KUKA KRL program: EPS_2_25694_LG03A_A_20260223033041.src

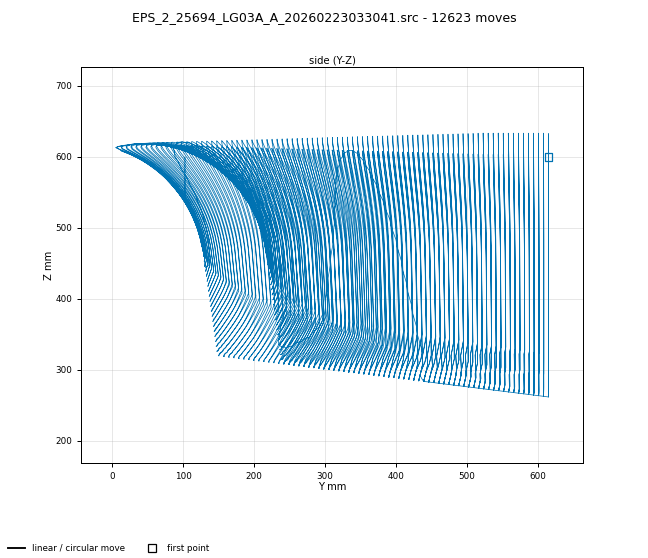
[picture p0: tool path of EPS_2_25694_LG03A_A_20260223033041.src, 12623 of 12625 moves have a stored position in this frame; points joined in program order, loops and branches not executed]
&ACCESS RVP
&REL 4
&COMMENT QRS 19112012
&PARAM EDITMASK = *
DEF PART()
EXT BAS (BAS_COMMAND :IN,REAL :IN )
INT I
BAS (#INITMOV,0 )

;KUKA QRS Post kuka4.cps  Date:22-06-2017 !

File_ID=3042

QRS_PRE_INIT()

;Init var - Until changes are made in qrs_pre_init
Outlet_Square_prg=0
Inlet_1_Square_prg=0
Inlet_2_Square_prg=0
Inlet_3_Square_prg=0
Inlet_4_Square_prg=0
Inlet_5_Square_prg=0

Outlet_1={X 0.000, Y 523.550, Z 484.000, B 0.000, E1 0.000 }
Inlet_1={X 0.000, Y 525.740, Z 454.000, B 0.000, E1 210.000 }
Outlet_1_type=299
Inlet_1_type=299
;QRS#1=Sidecore dimensions
;QRS#2=300-12" PVC SDR 35
;QRS#3=300-12" PVC SDR 35
;QRS#4=
;QRS#5=
;QRS#6=
;QRS#7=
;QRS#8=
;QRS#9=16M PSX
;QRS#10=16M PSX
;QRS#11=
;QRS#12=
;QRS#13=
;QRS#14=
;QRS#15=
;QRS#16=1220x127x914 3'
;QRS#17=EPS Height
;QRS#18=633,5
;QRS#19=*
;QRS#20= UPDATED VERSION 22-06-2017
;QRS#21=*
Outlet_Square=0150
Inlet_1_Square=0150
Inlet_2_Square=0
Inlet_3_Square=0
Inlet_4_Square=0
Inlet_5_Square=0
Mill_Square=1
Outlet_Square_Prg=206
Inlet_1_Square_prg=206

QRS_INIT()

$ADVANCE=5

; T1
PTP {E1 173.663,E2 173.663}
PTP {X 0,Y 615.411,A -85,B 0,C 180,E1 173.663,E2 173.663,E3 0,E4 0,E5 0,E6 0}
QRS_SPEED_INIT()
LIN {X 0,Y 615.411,Z 600,A -85,B 0,C 180,E1 173.663,E2 173.663,E3 0,E4 0,E5 0,E6 0} C_VEL
LIN {X 0,Y 615.411,Z 271.503,A -85,B 0,C 180,E1 173.663,E2 173.663} C_VEL
LIN {X 0,Y 615.411,Z 263.325,A -85,B 0,C 180,E1 173.663,E2 173.663} C_VEL
LIN {X 0,Y 615.409,Z 261.325,A -85,B 0,C 180,E1 173.477,E2 173.477} C_VEL
LIN {X 0,Y 615.462,Z 261.325,A -85,B 0,C 180,E1 170.802,E2 170.802} C_VEL
LIN {X 0,Y 615.44,Z 261.324,A -85,B 0,C 180,E1 168.14,E2 168.14} C_VEL
LIN {X 0,Y 615.434,Z 261.324,A -85,B 0,C 180,E1 166.084,E2 166.084} C_VEL
LIN {X 0,Y 615.412,Z 261.324,A -85,B 0,C 180,E1 163.59,E2 163.59} C_VEL
LIN {X 0,Y 615.421,Z 261.324,A -85,B 0,C 180,E1 161.353,E2 161.353} C_VEL
LIN {X 0,Y 615.489,Z 261.323,A -85,B 0,C 180,E1 158.57,E2 158.57} C_VEL
LIN {X 0,Y 615.417,Z 261.323,A -85,B 0,C 180,E1 155.727,E2 155.727} C_VEL
LIN {X 0,Y 615.419,Z 261.323,A -85,B 0,C 180,E1 153.554,E2 153.554} C_VEL
LIN {X 0,Y 615.479,Z 261.323,A -85,B 0,C 180,E1 150.595,E2 150.595} C_VEL
LIN {X 0,Y 615.45,Z 261.321,A -85,B 0,C 180,E1 148.314,E2 148.314} C_VEL
LIN {X 0,Y 615.424,Z 261.322,A -85,B 0,C 180,E1 145.976,E2 145.976} C_VEL
LIN {X 0,Y 615.426,Z 261.323,A -85,B 0,C 180,E1 143.573,E2 143.573} C_VEL
LIN {X 0,Y 615.491,Z 261.325,A -85,B 0,C 180,E1 140.936,E2 140.936} C_VEL
LIN {X 0,Y 615.47,Z 261.319,A -85,B 0,C 180,E1 138.527,E2 138.527} C_VEL
LIN {X 0,Y 615.425,Z 261.321,A -85,B 0,C 180,E1 136.008,E2 136.008} C_VEL
LIN {X 0,Y 615.428,Z 261.321,A -85,B 0,C 180,E1 133.994,E2 133.994} C_VEL
LIN {X 0,Y 615.442,Z 261.323,A -85,B 0,C 180,E1 131.477,E2 131.477} C_VEL
LIN {X 0,Y 615.495,Z 261.322,A -85,B 0,C 180,E1 128.903,E2 128.903} C_VEL
LIN {X 0,Y 615.453,Z 261.318,A -85,B 0,C 180,E1 126.426,E2 126.426} C_VEL
LIN {X 0,Y 615.431,Z 261.32,A -85,B 0,C 180,E1 124.025,E2 124.025} C_VEL
LIN {X 0,Y 615.487,Z 261.328,A -85,B 0,C 180,E1 121.09,E2 121.09} C_VEL
LIN {X 0,Y 615.45,Z 261.318,A -85,B 0,C 180,E1 118.448,E2 118.448} C_VEL
LIN {X 0,Y 615.452,Z 261.317,A -85,B 0,C 180,E1 116.445,E2 116.445} C_VEL
LIN {X 0,Y 615.435,Z 261.32,A -85,B 0,C 180,E1 114.002,E2 114.002} C_VEL
LIN {X 0,Y 615.47,Z 261.324,A -85,B 0,C 180,E1 111.432,E2 111.432} C_VEL
LIN {X 0,Y 615.464,Z 261.315,A -85,B 0,C 180,E1 108.605,E2 108.605} C_VEL
LIN {X 0,Y 615.449,Z 261.317,A -85,B 0,C 180,E1 106.426,E2 106.426} C_VEL
LIN {X 0,Y 615.444,Z 261.321,A -85,B 0,C 180,E1 103.875,E2 103.875} C_VEL
LIN {X 0,Y 615.484,Z 261.315,A -85,B 0,C 180,E1 100.898,E2 100.898} C_VEL
LIN {X 0,Y 615.455,Z 261.315,A -85,B 0,C 180,E1 98.537,E2 98.537} C_VEL
LIN {X 0,Y 615.456,Z 261.315,A -85,B 0,C 180,E1 96.557,E2 96.557} C_VEL
LIN {X 0,Y 615.456,Z 261.315,A -85,B 0,C 180,E1 94.585,E2 94.585} C_VEL
LIN {X 0,Y 615.46,Z 261.314,A -85,B 0,C 180,E1 92.618,E2 92.618} C_VEL
LIN {X 0,Y 615.462,Z 261.314,A -85,B 0,C 180,E1 90.655,E2 90.655} C_VEL
LIN {X 0,Y 615.447,Z 261.32,A -85,B 0,C 180,E1 88.037,E2 88.037} C_VEL
LIN {X 0,Y 615.497,Z 261.323,A -85,B 0,C 180,E1 85.416,E2 85.416} C_VEL
LIN {X 0,Y 615.471,Z 261.312,A -85,B 0,C 180,E1 82.785,E2 82.785} C_VEL
LIN {X 0,Y 615.448,Z 261.483,A -85,B 0,C 180,E1 82.248,E2 82.248} C_VEL
LIN {X 0,Y 615.472,Z 281.565,A -85,B 0,C 180,E1 79.64,E2 79.64} C_VEL
LIN {X 0,Y 615.452,Z 293.149,A -85,B 0,C 180,E1 78.181,E2 78.181} C_VEL
LIN {X 0,Y 615.487,Z 458.004,A -85,B 0,C 180,E1 76.19,E2 76.19} C_VEL
LIN {X 0,Y 615.486,Z 473.487,A -85,B 0,C 180,E1 75.866,E2 75.866} C_VEL
LIN {X 0,Y 615.481,Z 488.594,A -85,B 0,C 180,E1 75.409,E2 75.409} C_VEL
LIN {X 0,Y 615.487,Z 502.357,A -85,B 0,C 180,E1 74.859,E2 74.859} C_VEL
LIN {X 0,Y 615.489,Z 515.954,A -85,B 0,C 180,E1 74.181,E2 74.181} C_VEL
LIN {X 0,Y 615.497,Z 528.53,A -85,B 0,C 180,E1 73.414,E2 73.414} C_VEL
LIN {X 0,Y 615.496,Z 540.263,A -85,B 0,C 180,E1 72.559,E2 72.559} C_VEL
LIN {X 0,Y 615.497,Z 551.874,A -85,B 0,C 180,E1 71.551,E2 71.551} C_VEL
LIN {X 0,Y 615.496,Z 562.114,A -85,B 0,C 180,E1 70.49,E2 70.49} C_VEL
LIN {X 0,Y 615.493,Z 570.715,A -85,B 0,C 180,E1 69.436,E2 69.436} C_VEL
LIN {X 0,Y 615.498,Z 579.036,A -85,B 0,C 180,E1 68.217,E2 68.217} C_VEL
LIN {X 0,Y 615.494,Z 585.106,A -85,B 0,C 180,E1 67.157,E2 67.157} C_VEL
LIN {X 0,Y 615.492,Z 590.575,A -85,B 0,C 180,E1 65.986,E2 65.986} C_VEL
LIN {X 0,Y 615.498,Z 594.352,A -85,B 0,C 180,E1 65.01,E2 65.01} C_VEL
LIN {X 0,Y 615.49,Z 598.605,A -85,B 0,C 180,E1 63.557,E2 63.557} C_VEL
LIN {X 0,Y 615.493,Z 601.396,A -85,B 0,C 180,E1 62.086,E2 62.086} C_VEL
LIN {X 0,Y 615.496,Z 602.743,A -85,B 0,C 180,E1 60.595,E2 60.595} C_VEL
LIN {X 0,Y 615.496,Z 602.613,A -85,B 0,C 180,E1 59.082,E2 59.082} C_VEL
LIN {X 0,Y 615.49,Z 601.149,A -85,B 0,C 180,E1 57.665,E2 57.665} C_VEL
LIN {X 0,Y 615.491,Z 598.842,A -85,B 0,C 180,E1 56.462,E2 56.462} C_VEL
LIN {X 0,Y 615.499,Z 595.27,A -85,B 0,C 180,E1 55.187,E2 55.187} C_VEL
LIN {X 0,Y 615.497,Z 590.342,A -85,B 0,C 180,E1 53.87,E2 53.87} C_VEL
LIN {X 0,Y 615.497,Z 584.083,A -85,B 0,C 180,E1 52.567,E2 52.567} C_VEL
LIN {X 0,Y 615.493,Z 576.583,A -85,B 0,C 180,E1 51.307,E2 51.307} C_VEL
LIN {X 0,Y 615.494,Z 567.668,A -85,B 0,C 180,E1 50.08,E2 50.08} C_VEL
LIN {X 0,Y 615.494,Z 558.54,A -85,B 0,C 180,E1 49.026,E2 49.026} C_VEL
LIN {X 0,Y 615.494,Z 548.798,A -85,B 0,C 180,E1 48.07,E2 48.07} C_VEL
LIN {X 0,Y 615.496,Z 537.414,A -85,B 0,C 180,E1 47.125,E2 47.125} C_VEL
LIN {X 0,Y 615.498,Z 525.333,A -85,B 0,C 180,E1 46.285,E2 46.285} C_VEL
LIN {X 0,Y 615.485,Z 512.772,A -85,B 0,C 180,E1 45.558,E2 45.558} C_VEL
LIN {X 0,Y 615.493,Z 499.631,A -85,B 0,C 180,E1 44.934,E2 44.934} C_VEL
LIN {X 0,Y 615.49,Z 485.257,A -85,B 0,C 180,E1 44.392,E2 44.392} C_VEL
LIN {X 0,Y 615.492,Z 469.545,A -85,B 0,C 180,E1 43.952,E2 43.952} C_VEL
LIN {X 0,Y 615.492,Z 454.254,A -85,B 0,C 180,E1 43.667,E2 43.667} C_VEL
LIN {X 0,Y 615.466,Z 292.857,A -85,B 0,C 180,E1 41.719,E2 41.719} C_VEL
LIN {X 0,Y 615.478,Z 270.989,A -85,B 0,C 180,E1 38.903,E2 38.903} C_VEL
LIN {X 0,Y 615.477,Z 261.311,A -85,B 0,C 180,E1 37.626,E2 37.626} C_VEL
LIN {X 0,Y 615.484,Z 261.319,A -85,B 0,C 180,E1 34.702,E2 34.702} C_VEL
LIN {X 0,Y 615.486,Z 261.323,A -85,B 0,C 180,E1 32.333,E2 32.333} C_VEL
LIN {X 0,Y 615.485,Z 261.308,A -85,B 0,C 180,E1 29.405,E2 29.405} C_VEL
LIN {X 0,Y 615.482,Z 261.324,A -85,B 0,C 180,E1 26.443,E2 26.443} C_VEL
LIN {X 0,Y 615.482,Z 261.309,A -85,B 0,C 180,E1 23.555,E2 23.555} C_VEL
LIN {X 0,Y 615.481,Z 261.324,A -85,B 0,C 180,E1 20.559,E2 20.559} C_VEL
LIN {X 0,Y 615.46,Z 261.315,A -85,B 0,C 180,E1 17.956,E2 17.956} C_VEL
LIN {X 0,Y 615.492,Z 261.313,A -85,B 0,C 180,E1 15.225,E2 15.225} C_VEL
LIN {X 0,Y 615.469,Z 261.321,A -85,B 0,C 180,E1 12.529,E2 12.529} C_VEL
LIN {X 0,Y 615.461,Z 261.314,A -85,B 0,C 180,E1 9.861,E2 9.861} C_VEL
LIN {X 0,Y 615.494,Z 261.317,A -85,B 0,C 180,E1 7.214,E2 7.214} C_VEL
LIN {X 0,Y 615.459,Z 261.321,A -85,B 0,C 180,E1 4.584,E2 4.584} C_VEL
LIN {X 0,Y 615.454,Z 261.315,A -85,B 0,C 180,E1 1.962,E2 1.962} C_VEL
LIN {X 0,Y 615.494,Z 261.317,A -85,B 0,C 180,E1 -0.655,E2 -0.655} C_VEL
LIN {X 0,Y 615.454,Z 261.322,A -85,B 0,C 180,E1 -3.274,E2 -3.274} C_VEL
LIN {X 0,Y 615.454,Z 261.322,A -85,B 0,C 180,E1 -5.242,E2 -5.242} C_VEL
LIN {X 0,Y 615.452,Z 261.323,A -85,B 0,C 180,E1 -7.217,E2 -7.217} C_VEL
LIN {X 0,Y 615.45,Z 261.323,A -85,B 0,C 180,E1 -9.2,E2 -9.2} C_VEL
LIN {X 0,Y 615.447,Z 261.322,A -85,B 0,C 180,E1 -11.195,E2 -11.195} C_VEL
LIN {X 0,Y 615.443,Z 261.322,A -85,B 0,C 180,E1 -13.203,E2 -13.203} C_VEL
LIN {X 0,Y 615.438,Z 261.322,A -85,B 0,C 180,E1 -15.228,E2 -15.228} C_VEL
LIN {X 0,Y 615.433,Z 261.322,A -85,B 0,C 180,E1 -17.273,E2 -17.273} C_VEL
LIN {X 0,Y 615.427,Z 261.322,A -85,B 0,C 180,E1 -19.341,E2 -19.341} C_VEL
LIN {X 0,Y 615.423,Z 261.322,A -85,B 0,C 180,E1 -21.435,E2 -21.435} C_VEL
LIN {X 0,Y 615.446,Z 261.322,A -85,B 0,C 180,E1 -24.003,E2 -24.003} C_VEL
LIN {X 0,Y 615.492,Z 261.327,A -85,B 0,C 180,E1 -26.445,E2 -26.445} C_VEL
LIN {X 0,Y 615.462,Z 261.325,A -85,B 0,C 180,E1 -28.66,E2 -28.66} C_VEL
LIN {X 0,Y 615.419,Z 261.325,A -85,B 0,C 180,E1 -31.078,E2 -31.078} C_VEL
LIN {X 0,Y 615.411,Z 261.325,A -85,B 0,C 180,E1 -33.241,E2 -33.241} C_VEL
LIN {X 0,Y 615.435,Z 261.326,A -85,B 0,C 180,E1 -35.829,E2 -35.829} C_VEL
LIN {X 0,Y 615.473,Z 261.325,A -85,B 0,C 180,E1 -38.07,E2 -38.07} C_VEL
LIN {X 0,Y 615.452,Z 261.323,A -85,B 0,C 180,E1 -40.61,E2 -40.61} C_VEL
LIN {X 0,Y 615.422,Z 261.323,A -85,B 0,C 180,E1 -43.043,E2 -43.043} C_VEL
LIN {X 0,Y 615.422,Z 261.322,A -85,B 0,C 180,E1 -45.075,E2 -45.075} C_VEL
LIN {X 0,Y 615.446,Z 261.324,A -85,B 0,C 180,E1 -47.645,E2 -47.645} C_VEL
LIN {X 0,Y 615.491,Z 261.319,A -85,B 0,C 180,E1 -50.252,E2 -50.252} C_VEL
LIN {X 0,Y 615.439,Z 261.32,A -85,B 0,C 180,E1 -52.756,E2 -52.756} C_VEL
LIN {X 0,Y 615.431,Z 261.322,A -85,B 0,C 180,E1 -55.183,E2 -55.183} C_VEL
LIN {X 0,Y 615.472,Z 261.324,A -85,B 0,C 180,E1 -57.672,E2 -57.672} C_VEL
LIN {X 0,Y 615.452,Z 261.317,A -85,B 0,C 180,E1 -60.593,E2 -60.593} C_VEL
LIN {X 0,Y 615.439,Z 261.319,A -85,B 0,C 180,E1 -62.964,E2 -62.964} C_VEL
LIN {X 0,Y 615.441,Z 261.447,A -85,B 0,C 180,E1 -64.936,E2 -64.936} C_VEL
LIN {X 0,Y 615.482,Z 284.085,A -85,B 0,C 180,E1 -67.53,E2 -67.53} C_VEL
LIN {X 0,Y 615.49,Z 308.883,A -85,B 0,C 180,E1 -70.316,E2 -70.316} C_VEL
LIN {X 0,Y 615.488,Z 322.077,A -85,B 0,C 180,E1 -71.762,E2 -71.762} C_VEL
LIN {X 0,Y 615.487,Z 488.142,A -85,B 0,C 180,E1 -73.768,E2 -73.768} C_VEL
LIN {X 0,Y 615.49,Z 503.738,A -85,B 0,C 180,E1 -74.096,E2 -74.096} C_VEL
LIN {X 0,Y 615.48,Z 519.068,A -85,B 0,C 180,E1 -74.562,E2 -74.562} C_VEL
LIN {X 0,Y 615.492,Z 532.768,A -85,B 0,C 180,E1 -75.113,E2 -75.113} C_VEL
LIN {X 0,Y 615.494,Z 547.053,A -85,B 0,C 180,E1 -75.834,E2 -75.834} C_VEL
LIN {X 0,Y 615.497,Z 559.907,A -85,B 0,C 180,E1 -76.632,E2 -76.632} C_VEL
LIN {X 0,Y 615.495,Z 572.262,A -85,B 0,C 180,E1 -77.554,E2 -77.554} C_VEL
LIN {X 0,Y 615.495,Z 582.612,A -85,B 0,C 180,E1 -78.474,E2 -78.474} C_VEL
LIN {X 0,Y 615.495,Z 592.189,A -85,B 0,C 180,E1 -79.474,E2 -79.474} C_VEL
LIN {X 0,Y 615.494,Z 601.581,A -85,B 0,C 180,E1 -80.636,E2 -80.636} C_VEL
LIN {X 0,Y 615.495,Z 609.384,A -85,B 0,C 180,E1 -81.795,E2 -81.795} C_VEL
LIN {X 0,Y 615.496,Z 616.608,A -85,B 0,C 180,E1 -83.102,E2 -83.102} C_VEL
LIN {X 0,Y 615.499,Z 622.438,A -85,B 0,C 180,E1 -84.431,E2 -84.431} C_VEL
LIN {X 0,Y 615.491,Z 625.861,A -85,B 0,C 180,E1 -85.416,E2 -85.416} C_VEL
LIN {X 0,Y 615.492,Z 629.319,A -85,B 0,C 180,E1 -86.727,E2 -86.727} C_VEL
LIN {X 0,Y 615.497,Z 631.594,A -85,B 0,C 180,E1 -88.037,E2 -88.037} C_VEL
LIN {X 0,Y 615.493,Z 632.741,A -85,B 0,C 180,E1 -89.346,E2 -89.346} C_VEL
LIN {X 0,Y 615.493,Z 632.74,A -85,B 0,C 180,E1 -90.654,E2 -90.654} C_VEL
LIN {X 0,Y 615.497,Z 631.593,A -85,B 0,C 180,E1 -91.963,E2 -91.963} C_VEL
LIN {X 0,Y 615.492,Z 629.318,A -85,B 0,C 180,E1 -93.273,E2 -93.273} C_VEL
LIN {X 0,Y 615.491,Z 625.86,A -85,B 0,C 180,E1 -94.585,E2 -94.585} C_VEL
LIN {X 0,Y 615.49,Z 621.143,A -85,B 0,C 180,E1 -95.899,E2 -95.899} C_VEL
LIN {X 0,Y 615.495,Z 615.029,A -85,B 0,C 180,E1 -97.216,E2 -97.216} C_VEL
LIN {X 0,Y 615.49,Z 607.332,A -85,B 0,C 180,E1 -98.537,E2 -98.537} C_VEL
LIN {X 0,Y 615.495,Z 599.113,A -85,B 0,C 180,E1 -99.696,E2 -99.696} C_VEL
LIN {X 0,Y 615.497,Z 588.897,A -85,B 0,C 180,E1 -100.892,E2 -100.892} C_VEL
LIN {X 0,Y 615.495,Z 579.067,A -85,B 0,C 180,E1 -101.861,E2 -101.861} C_VEL
LIN {X 0,Y 615.498,Z 566.947,A -85,B 0,C 180,E1 -102.865,E2 -102.865} C_VEL
LIN {X 0,Y 615.498,Z 554.798,A -85,B 0,C 180,E1 -103.705,E2 -103.705} C_VEL
LIN {X 0,Y 615.484,Z 541.38,A -85,B 0,C 180,E1 -104.472,E2 -104.472} C_VEL
LIN {X 0,Y 615.495,Z 526.849,A -85,B 0,C 180,E1 -105.141,E2 -105.141} C_VEL
LIN {X 0,Y 615.484,Z 512.618,A -85,B 0,C 180,E1 -105.65,E2 -105.65} C_VEL
LIN {X 0,Y 615.499,Z 498.131,A -85,B 0,C 180,E1 -106.036,E2 -106.036} C_VEL
LIN {X 0,Y 615.487,Z 483.544,A -85,B 0,C 180,E1 -106.298,E2 -106.298} C_VEL
LIN {X 0,Y 615.489,Z 321.745,A -85,B 0,C 180,E1 -108.258,E2 -108.258} C_VEL
LIN {X 0,Y 615.49,Z 296.393,A -85,B 0,C 180,E1 -111.081,E2 -111.081} C_VEL
LIN {X 0,Y 615.495,Z 270.582,A -85,B 0,C 180,E1 -114.01,E2 -114.01} C_VEL
LIN {X 0,Y 615.441,Z 261.318,A -85,B 0,C 180,E1 -115.1,E2 -115.1} C_VEL
LIN {X 0,Y 615.489,Z 261.317,A -85,B 0,C 180,E1 -117.915,E2 -117.915} C_VEL
LIN {X 0,Y 615.498,Z 261.324,A -85,B 0,C 180,E1 -120.159,E2 -120.159} C_VEL
LIN {X 0,Y 615.465,Z 261.323,A -85,B 0,C 180,E1 -122.458,E2 -122.458} C_VEL
LIN {X 0,Y 615.439,Z 261.32,A -85,B 0,C 180,E1 -124.818,E2 -124.818} C_VEL
LIN {X 0,Y 615.443,Z 261.318,A -85,B 0,C 180,E1 -127.245,E2 -127.245} C_VEL
LIN {X 0,Y 615.498,Z 261.326,A -85,B 0,C 180,E1 -130.09,E2 -130.09} C_VEL
LIN {X 0,Y 615.463,Z 261.323,A -85,B 0,C 180,E1 -132.354,E2 -132.354} C_VEL
LIN {X 0,Y 615.433,Z 261.32,A -85,B 0,C 180,E1 -134.926,E2 -134.926} C_VEL
LIN {X 0,Y 615.433,Z 261.32,A -85,B 0,C 180,E1 -136.957,E2 -136.957} C_VEL
LIN {X 0,Y 615.457,Z 261.317,A -85,B 0,C 180,E1 -139.391,E2 -139.391} C_VEL
LIN {X 0,Y 615.481,Z 261.328,A -85,B 0,C 180,E1 -141.988,E2 -141.988} C_VEL
LIN {X 0,Y 615.446,Z 261.323,A -85,B 0,C 180,E1 -144.381,E2 -144.381} C_VEL
LIN {X 0,Y 615.428,Z 261.321,A -85,B 0,C 180,E1 -146.76,E2 -146.76} C_VEL
LIN {X 0,Y 615.435,Z 261.32,A -85,B 0,C 180,E1 -149.077,E2 -149.077} C_VEL
LIN {X 0,Y 615.484,Z 261.318,A -85,B 0,C 180,E1 -151.549,E2 -151.549} C_VEL
LIN {X 0,Y 615.443,Z 261.323,A -85,B 0,C 180,E1 -154.282,E2 -154.282} C_VEL
LIN {X 0,Y 615.43,Z 261.323,A -85,B 0,C 180,E1 -156.441,E2 -156.441} C_VEL
LIN {X 0,Y 615.424,Z 261.323,A -85,B 0,C 180,E1 -158.565,E2 -158.565} C_VEL
LIN {X 0,Y 615.422,Z 261.322,A -85,B 0,C 180,E1 -160.659,E2 -160.659} C_VEL
LIN {X 0,Y 615.47,Z 261.321,A -85,B 0,C 180,E1 -163.412,E2 -163.412} C_VEL
LIN {X 0,Y 615.443,Z 261.324,A -85,B 0,C 180,E1 -166.124,E2 -166.124} C_VEL
LIN {X 0,Y 615.44,Z 261.324,A -85,B 0,C 180,E1 -168.137,E2 -168.137} C_VEL
LIN {X 0,Y 615.437,Z 261.324,A -85,B 0,C 180,E1 -170.136,E2 -170.136} C_VEL
LIN {X 0,Y 615.436,Z 261.324,A -85,B 0,C 180,E1 -172.123,E2 -172.123} C_VEL
LIN {X 0,Y 615.436,Z 261.324,A -85,B 0,C 180,E1 -174.1,E2 -174.1} C_VEL
LIN {X 0,Y 615.436,Z 261.324,A -85,B 0,C 180,E1 -176.07,E2 -176.07} C_VEL
LIN {X 0,Y 615.437,Z 261.325,A -85,B 0,C 180,E1 -178.036,E2 -178.036} C_VEL
LIN {X 0,Y 615.437,Z 261.325,A -85,B 0,C 180,E1 -179.999,E2 -179.999} C_VEL
LIN {X 0,Y 615.439,Z 261.325,A -85,B 0,C 180,E1 -181.962,E2 -181.962} C_VEL
LIN {X 0,Y 615.44,Z 261.325,A -85,B 0,C 180,E1 -183.928,E2 -183.928} C_VEL
LIN {X 0,Y 615.409,Z 261.325,A -85,B 0,C 180,E1 -186.523,E2 -186.523} C_VEL
LIN {X 0,Y 614.767,Z 261.474,A -85,B 0,C 180,E1 -187.069,E2 -187.069} C_VEL
LIN {X 0,Y 611.966,Z 261.877,A -85,B 0,C 180,E1 -187.955,E2 -187.955} C_VEL
LIN {X 0,Y 609.577,Z 262.192,A -85,B 0,C 180,E1 -188.668,E2 -188.668} C_VEL
LIN {X 0,Y 608.529,Z 262.313,A -85,B 0,C 180,E1 -189.218,E2 -189.218} C_VEL
LIN {X 0,Y 608.433,Z 262.321,A -85,B 0,C 180,E1 -189.404,E2 -189.404} C_VEL
LIN {X 0,Y 608.414,Z 262.319,A -85,B 0,C 180,E1 -191.999,E2 -191.999} C_VEL
LIN {X 0,Y 608.405,Z 262.319,A -85,B 0,C 180,E1 -194.038,E2 -194.038} C_VEL
LIN {X 0,Y 608.384,Z 262.32,A -85,B 0,C 180,E1 -196.506,E2 -196.506} C_VEL
LIN {X 0,Y 608.423,Z 262.319,A -85,B 0,C 180,E1 -198.869,E2 -198.869} C_VEL
LIN {X 0,Y 608.445,Z 262.317,A -85,B 0,C 180,E1 -201.691,E2 -201.691} C_VEL
LIN {X 0,Y 608.408,Z 262.319,A -85,B 0,C 180,E1 -204.571,E2 -204.571} C_VEL
LIN {X 0,Y 608.467,Z 262.32,A -85,B 0,C 180,E1 -207.207,E2 -207.207} C_VEL
LIN {X 0,Y 608.402,Z 262.319,A -85,B 0,C 180,E1 -209.962,E2 -209.962} C_VEL
LIN {X 0,Y 608.415,Z 262.317,A -85,B 0,C 180,E1 -212.095,E2 -212.095} C_VEL
LIN {X 0,Y 608.417,Z 262.323,A -85,B 0,C 180,E1 -214.902,E2 -214.902} C_VEL
LIN {X 0,Y 608.433,Z 262.316,A -85,B 0,C 180,E1 -217.747,E2 -217.747} C_VEL
LIN {X 0,Y 608.414,Z 262.318,A -85,B 0,C 180,E1 -220.326,E2 -220.326} C_VEL
LIN {X 0,Y 608.443,Z 262.322,A -85,B 0,C 180,E1 -222.958,E2 -222.958} C_VEL
LIN {X 0,Y 608.413,Z 262.318,A -85,B 0,C 180,E1 -225.738,E2 -225.738} C_VEL
LIN {X 0,Y 608.413,Z 262.317,A -85,B 0,C 180,E1 -227.935,E2 -227.935} C_VEL
LIN {X 0,Y 608.43,Z 262.321,A -85,B 0,C 180,E1 -230.704,E2 -230.704} C_VEL
LIN {X 0,Y 608.46,Z 262.32,A -85,B 0,C 180,E1 -233.086,E2 -233.086} C_VEL
LIN {X 0,Y 608.452,Z 262.314,A -85,B 0,C 180,E1 -235.53,E2 -235.53} C_VEL
LIN {X 0,Y 608.425,Z 262.316,A -85,B 0,C 180,E1 -237.904,E2 -237.904} C_VEL
LIN {X 0,Y 608.421,Z 262.317,A -85,B 0,C 180,E1 -240.218,E2 -240.218} C_VEL
LIN {X 0,Y 608.477,Z 262.319,A -85,B 0,C 180,E1 -242.789,E2 -242.789} C_VEL
LIN {X 0,Y 608.435,Z 262.314,A -85,B 0,C 180,E1 -245.852,E2 -245.852} C_VEL
LIN {X 0,Y 608.44,Z 262.317,A -85,B 0,C 180,E1 -248.308,E2 -248.308} C_VEL
LIN {X 0,Y 608.451,Z 262.315,A -85,B 0,C 180,E1 -251.283,E2 -251.283} C_VEL
LIN {X 0,Y 608.42,Z 262.316,A -85,B 0,C 180,E1 -253.905,E2 -253.905} C_VEL
LIN {X 0,Y 608.461,Z 262.321,A -85,B 0,C 180,E1 -256.644,E2 -256.644} C_VEL
LIN {X 0,Y 608.443,Z 262.315,A -85,B 0,C 180,E1 -259.35,E2 -259.35} C_VEL
LIN {X 0,Y 608.444,Z 262.315,A -85,B 0,C 180,E1 -262.033,E2 -262.033} C_VEL
LIN {X 0,Y 608.469,Z 262.32,A -85,B 0,C 180,E1 -264.698,E2 -264.698} C_VEL
LIN {X 0,Y 608.453,Z 262.313,A -85,B 0,C 180,E1 -267.352,E2 -267.352} C_VEL
LIN {X 0,Y 608.442,Z 262.316,A -85,B 0,C 180,E1 -270,E2 -270} C_VEL
LIN {X 0,Y 608.484,Z 262.317,A -85,B 0,C 180,E1 -272.648,E2 -272.648} C_VEL
LIN {X 0,Y 608.446,Z 262.314,A -85,B 0,C 180,E1 -275.302,E2 -275.302} C_VEL
LIN {X 0,Y 608.431,Z 262.317,A -85,B 0,C 180,E1 -277.591,E2 -277.591} C_VEL
LIN {X 0,Y 608.559,Z 276.552,A -85,B 0,C 180,E1 -279.472,E2 -279.472} C_VEL
LIN {X 0,Y 608.519,Z 292.986,A -85,B 0,C 180,E1 -281.602,E2 -281.602} C_VEL
LIN {X 0,Y 608.721,Z 316.53,A -85,B 0,C 180,E1 -281.895,E2 -281.895} C_VEL
LIN {X 0,Y 608.666,Z 458.242,A -85,B 0,C 180,E1 -283.628,E2 -283.628} C_VEL
LIN {X 0,Y 608.667,Z 474.141,A -85,B 0,C 180,E1 -283.968,E2 -283.968} C_VEL
LIN {X 0,Y 608.618,Z 489.893,A -85,B 0,C 180,E1 -284.46,E2 -284.46} C_VEL
LIN {X 0,Y 608.596,Z 504.382,A -85,B 0,C 180,E1 -285.059,E2 -285.059} C_VEL
LIN {X 0,Y 608.562,Z 517.647,A -85,B 0,C 180,E1 -285.746,E2 -285.746} C_VEL
LIN {X 0,Y 608.546,Z 530.554,A -85,B 0,C 180,E1 -286.561,E2 -286.561} C_VEL
LIN {X 0,Y 608.508,Z 542.604,A -85,B 0,C 180,E1 -287.474,E2 -287.474} C_VEL
LIN {X 0,Y 608.493,Z 553.997,A -85,B 0,C 180,E1 -288.503,E2 -288.503} C_VEL
LIN {X 0,Y 608.467,Z 563.931,A -85,B 0,C 180,E1 -289.569,E2 -289.569} C_VEL
LIN {X 0,Y 608.46,Z 573.467,A -85,B 0,C 180,E1 -290.79,E2 -290.79} C_VEL
LIN {X 0,Y 608.453,Z 581.573,A -85,B 0,C 180,E1 -292.048,E2 -292.048} C_VEL
LIN {X 0,Y 608.434,Z 587.306,A -85,B 0,C 180,E1 -293.124,E2 -293.124} C_VEL
LIN {X 0,Y 608.427,Z 591.904,A -85,B 0,C 180,E1 -294.147,E2 -294.147} C_VEL
LIN {X 0,Y 608.437,Z 596.043,A -85,B 0,C 180,E1 -295.301,E2 -295.301} C_VEL
LIN {X 0,Y 608.422,Z 599.973,A -85,B 0,C 180,E1 -296.775,E2 -296.775} C_VEL
LIN {X 0,Y 608.434,Z 602.436,A -85,B 0,C 180,E1 -298.267,E2 -298.267} C_VEL
LIN {X 0,Y 608.447,Z 603.444,A -85,B 0,C 180,E1 -299.78,E2 -299.78} C_VEL
LIN {X 0,Y 608.435,Z 602.948,A -85,B 0,C 180,E1 -301.317,E2 -301.317} C_VEL
LIN {X 0,Y 608.416,Z 601.474,A -85,B 0,C 180,E1 -302.519,E2 -302.519} C_VEL
LIN {X 0,Y 608.433,Z 598.145,A -85,B 0,C 180,E1 -304.073,E2 -304.073} C_VEL
LIN {X 0,Y 608.425,Z 594.42,A -85,B 0,C 180,E1 -305.278,E2 -305.278} C_VEL
LIN {X 0,Y 608.449,Z 589.516,A -85,B 0,C 180,E1 -306.501,E2 -306.501} C_VEL
LIN {X 0,Y 608.439,Z 583.238,A -85,B 0,C 180,E1 -307.747,E2 -307.747} C_VEL
LIN {X 0,Y 608.469,Z 575.898,A -85,B 0,C 180,E1 -308.943,E2 -308.943} C_VEL
LIN {X 0,Y 608.468,Z 567.519,A -85,B 0,C 180,E1 -310.084,E2 -310.084} C_VEL
LIN {X 0,Y 608.472,Z 558.024,A -85,B 0,C 180,E1 -311.174,E2 -311.174} C_VEL
LIN {X 0,Y 608.498,Z 547.442,A -85,B 0,C 180,E1 -312.199,E2 -312.199} C_VEL
LIN {X 0,Y 608.545,Z 536.009,A -85,B 0,C 180,E1 -313.133,E2 -313.133} C_VEL
LIN {X 0,Y 608.561,Z 523.952,A -85,B 0,C 180,E1 -313.965,E2 -313.965} C_VEL
LIN {X 0,Y 608.568,Z 511.052,A -85,B 0,C 180,E1 -314.703,E2 -314.703} C_VEL
LIN {X 0,Y 608.63,Z 496.659,A -85,B 0,C 180,E1 -315.369,E2 -315.369} C_VEL
LIN {X 0,Y 608.641,Z 482.482,A -85,B 0,C 180,E1 -315.881,E2 -315.881} C_VEL
LIN {X 0,Y 608.669,Z 467.061,A -85,B 0,C 180,E1 -316.291,E2 -316.291} C_VEL
LIN {X 0,Y 608.695,Z 451.014,A -85,B 0,C 180,E1 -316.567,E2 -316.567} C_VEL
LIN {X 0,Y 608.686,Z 293.883,A -85,B 0,C 180,E1 -318.472,E2 -318.472} C_VEL
LIN {X 0,Y 608.511,Z 292.853,A -85,B 0,C 180,E1 -318.5,E2 -318.5} C_VEL
LIN {X 0,Y 608.574,Z 271.809,A -85,B 0,C 180,E1 -321.24,E2 -321.24} C_VEL
LIN {X 0,Y 608.452,Z 262.314,A -85,B 0,C 180,E1 -322.517,E2 -322.517} C_VEL
LIN {X 0,Y 608.471,Z 262.314,A -85,B 0,C 180,E1 -325.089,E2 -325.089} C_VEL
LIN {X 0,Y 608.462,Z 262.315,A -85,B 0,C 180,E1 -327.907,E2 -327.907} C_VEL
LIN {X 0,Y 608.454,Z 262.313,A -85,B 0,C 180,E1 -330.222,E2 -330.222} C_VEL
LIN {X 0,Y 608.474,Z 262.311,A -85,B 0,C 180,E1 -332.791,E2 -332.791} C_VEL
LIN {X 0,Y 608.443,Z 262.324,A -85,B 0,C 180,E1 -335.43,E2 -335.43} C_VEL
LIN {X 0,Y 608.463,Z 262.311,A -85,B 0,C 180,E1 -338.31,E2 -338.31} C_VEL
LIN {X 0,Y 608.462,Z 262.322,A -85,B 0,C 180,E1 -341.282,E2 -341.282} C_VEL
LIN {X 0,Y 608.438,Z 262.315,A -85,B 0,C 180,E1 -343.907,E2 -343.907} C_VEL
LIN {X 0,Y 608.461,Z 262.314,A -85,B 0,C 180,E1 -346.645,E2 -346.645} C_VEL
LIN {X 0,Y 608.451,Z 262.319,A -85,B 0,C 180,E1 -349.351,E2 -349.351} C_VEL
LIN {X 0,Y 608.452,Z 262.312,A -85,B 0,C 180,E1 -352.034,E2 -352.034} C_VEL
LIN {X 0,Y 608.469,Z 262.315,A -85,B 0,C 180,E1 -354.699,E2 -354.699} C_VEL
LIN {X 0,Y 608.452,Z 262.317,A -85,B 0,C 180,E1 -357.353,E2 -357.353} C_VEL
LIN {X 0,Y 608.444,Z 262.313,A -85,B 0,C 180,E1 -360.001,E2 -360.001} C_VEL
LIN {X 0,Y 608.484,Z 262.315,A -85,B 0,C 180,E1 -362.649,E2 -362.649} C_VEL
LIN {X 0,Y 608.433,Z 262.318,A -85,B 0,C 180,E1 -365.303,E2 -365.303} C_VEL
LIN {X 0,Y 608.419,Z 262.319,A -85,B 0,C 180,E1 -367.301,E2 -367.301} C_VEL
LIN {X 0,Y 608.421,Z 262.317,A -85,B 0,C 180,E1 -369.979,E2 -369.979} C_VEL
LIN {X 0,Y 608.47,Z 262.321,A -85,B 0,C 180,E1 -372.678,E2 -372.678} C_VEL
LIN {X 0,Y 608.427,Z 262.316,A -85,B 0,C 180,E1 -375.408,E2 -375.408} C_VEL
LIN {X 0,Y 608.407,Z 262.318,A -85,B 0,C 180,E1 -377.479,E2 -377.479} C_VEL
LIN {X 0,Y 608.406,Z 262.318,A -85,B 0,C 180,E1 -379.573,E2 -379.573} C_VEL
LIN {X 0,Y 608.423,Z 262.316,A -85,B 0,C 180,E1 -381.694,E2 -381.694} C_VEL
LIN {X 0,Y 608.431,Z 262.324,A -85,B 0,C 180,E1 -384.573,E2 -384.573} C_VEL
LIN {X 0,Y 608.405,Z 262.319,A -85,B 0,C 180,E1 -387.197,E2 -387.197} C_VEL
LIN {X 0,Y 608.397,Z 262.321,A -85,B 0,C 180,E1 -389.024,E2 -389.024} C_VEL
LIN {X 0,Y 608.396,Z 262.319,A -85,B 0,C 180,E1 -391.321,E2 -391.321} C_VEL
LIN {X 0,Y 608.415,Z 262.319,A -85,B 0,C 180,E1 -393.729,E2 -393.729} C_VEL
LIN {X 0,Y 608.429,Z 262.323,A -85,B 0,C 180,E1 -396.094,E2 -396.094} C_VEL
LIN {X 0,Y 608.399,Z 262.323,A -85,B 0,C 180,E1 -398.594,E2 -398.594} C_VEL
LIN {X 0,Y 608.389,Z 262.32,A -85,B 0,C 180,E1 -401.183,E2 -401.183} C_VEL
LIN {X 0,Y 608.416,Z 262.317,A -85,B 0,C 180,E1 -403.305,E2 -403.305} C_VEL
LIN {X 0,Y 608.458,Z 262.322,A -85,B 0,C 180,E1 -406.131,E2 -406.131} C_VEL
LIN {X 0,Y 608.406,Z 262.319,A -85,B 0,C 180,E1 -408.821,E2 -408.821} C_VEL
LIN {X 0,Y 608.454,Z 262.319,A -85,B 0,C 180,E1 -411.762,E2 -411.762} C_VEL
LIN {X 0,Y 608.417,Z 262.317,A -85,B 0,C 180,E1 -414.722,E2 -414.722} C_VEL
LIN {X 0,Y 608.425,Z 262.316,A -85,B 0,C 180,E1 -417.12,E2 -417.12} C_VEL
LIN {X 0,Y 608.476,Z 262.317,A -85,B 0,C 180,E1 -420.027,E2 -420.027} C_VEL
LIN {X 0,Y 608.421,Z 262.317,A -85,B 0,C 180,E1 -422.804,E2 -422.804} C_VEL
LIN {X 0,Y 608.448,Z 262.455,A -85,B 0,C 180,E1 -424.746,E2 -424.746} C_VEL
LIN {X 0,Y 608.665,Z 274.55,A -85,B 0,C 180,E1 -426.164,E2 -426.164} C_VEL
LIN {X 0,Y 608.595,Z 297.959,A -85,B 0,C 180,E1 -428.847,E2 -428.847} C_VEL
LIN {X 0,Y 608.574,Z 322.077,A -85,B 0,C 180,E1 -431.548,E2 -431.548} C_VEL
LIN {X 0,Y 608.727,Z 425.97,A -85,B 0,C 180,E1 -432.814,E2 -432.814} C_VEL
LIN {X 0,Y 608.682,Z 488.142,A -85,B 0,C 180,E1 -433.581,E2 -433.581} C_VEL
LIN {X 0,Y 608.65,Z 503.736,A -85,B 0,C 180,E1 -433.912,E2 -433.912} C_VEL
LIN {X 0,Y 608.618,Z 519.067,A -85,B 0,C 180,E1 -434.384,E2 -434.384} C_VEL
LIN {X 0,Y 608.606,Z 532.771,A -85,B 0,C 180,E1 -434.941,E2 -434.941} C_VEL
LIN {X 0,Y 608.575,Z 546.248,A -85,B 0,C 180,E1 -435.625,E2 -435.625} C_VEL
LIN {X 0,Y 608.554,Z 558.673,A -85,B 0,C 180,E1 -436.391,E2 -436.391} C_VEL
LIN {X 0,Y 608.528,Z 571.29,A -85,B 0,C 180,E1 -437.325,E2 -437.325} C_VEL
LIN {X 0,Y 608.496,Z 582.753,A -85,B 0,C 180,E1 -438.34,E2 -438.34} C_VEL
LIN {X 0,Y 608.476,Z 592.393,A -85,B 0,C 180,E1 -439.351,E2 -439.351} C_VEL
LIN {X 0,Y 608.477,Z 601.857,A -85,B 0,C 180,E1 -440.527,E2 -440.527} C_VEL
LIN {X 0,Y 608.455,Z 609.732,A -85,B 0,C 180,E1 -441.699,E2 -441.699} C_VEL
LIN {X 0,Y 608.441,Z 617.089,A -85,B 0,C 180,E1 -443.034,E2 -443.034} C_VEL
LIN {X 0,Y 608.449,Z 622.925,A -85,B 0,C 180,E1 -444.366,E2 -444.366} C_VEL
LIN {X 0,Y 608.427,Z 626.384,A -85,B 0,C 180,E1 -445.363,E2 -445.363} C_VEL
LIN {X 0,Y 608.421,Z 629.886,A -85,B 0,C 180,E1 -446.689,E2 -446.689} C_VEL
LIN {X 0,Y 608.442,Z 632.192,A -85,B 0,C 180,E1 -448.014,E2 -448.014} C_VEL
LIN {X 0,Y 608.436,Z 633.351,A -85,B 0,C 180,E1 -449.338,E2 -449.338} C_VEL
LIN {X 0,Y 608.436,Z 633.35,A -85,B 0,C 180,E1 -450.662,E2 -450.662} C_VEL
LIN {X 0,Y 608.442,Z 632.191,A -85,B 0,C 180,E1 -451.986,E2 -451.986} C_VEL
LIN {X 0,Y 608.421,Z 629.885,A -85,B 0,C 180,E1 -453.311,E2 -453.311} C_VEL
LIN {X 0,Y 608.427,Z 626.382,A -85,B 0,C 180,E1 -454.638,E2 -454.638} C_VEL
LIN {X 0,Y 608.431,Z 621.607,A -85,B 0,C 180,E1 -455.967,E2 -455.967} C_VEL
LIN {X 0,Y 608.458,Z 615.425,A -85,B 0,C 180,E1 -457.3,E2 -457.3} C_VEL
LIN {X 0,Y 608.465,Z 607.653,A -85,B 0,C 180,E1 -458.636,E2 -458.636} C_VEL
LIN {X 0,Y 608.471,Z 599.37,A -85,B 0,C 180,E1 -459.809,E2 -459.809} C_VEL
LIN {X 0,Y 608.492,Z 588.651,A -85,B 0,C 180,E1 -461.063,E2 -461.063} C_VEL
LIN {X 0,Y 608.522,Z 577.274,A -85,B 0,C 180,E1 -462.168,E2 -462.168} C_VEL
LIN {X 0,Y 608.548,Z 565.854,A -85,B 0,C 180,E1 -463.1,E2 -463.1} C_VEL
LIN {X 0,Y 608.563,Z 553.447,A -85,B 0,C 180,E1 -463.95,E2 -463.95} C_VEL
LIN {X 0,Y 608.569,Z 539.86,A -85,B 0,C 180,E1 -464.718,E2 -464.718} C_VEL
LIN {X 0,Y 608.633,Z 525.793,A -85,B 0,C 180,E1 -465.359,E2 -465.359} C_VEL
LIN {X 0,Y 608.636,Z 511.303,A -85,B 0,C 180,E1 -465.874,E2 -465.874} C_VEL
LIN {X 0,Y 608.689,Z 496.005,A -85,B 0,C 180,E1 -466.27,E2 -466.27} C_VEL
LIN {X 0,Y 608.688,Z 480.032,A -85,B 0,C 180,E1 -466.534,E2 -466.534} C_VEL
LIN {X 0,Y 608.683,Z 322.68,A -85,B 0,C 180,E1 -468.441,E2 -468.441} C_VEL
LIN {X 0,Y 608.541,Z 321.57,A -85,B 0,C 180,E1 -468.494,E2 -468.494} C_VEL
LIN {X 0,Y 608.62,Z 296.393,A -85,B 0,C 180,E1 -471.33,E2 -471.33} C_VEL
LIN {X 0,Y 608.683,Z 271.446,A -85,B 0,C 180,E1 -474.195,E2 -474.195} C_VEL
LIN {X 0,Y 608.448,Z 262.45,A -85,B 0,C 180,E1 -475.255,E2 -475.255} C_VEL
LIN {X 0,Y 608.443,Z 262.324,A -85,B 0,C 180,E1 -478.267,E2 -478.267} C_VEL
LIN {X 0,Y 608.453,Z 262.317,A -85,B 0,C 180,E1 -480.545,E2 -480.545} C_VEL
LIN {X 0,Y 608.43,Z 262.316,A -85,B 0,C 180,E1 -482.881,E2 -482.881} C_VEL
LIN {X 0,Y 608.421,Z 262.316,A -85,B 0,C 180,E1 -485.279,E2 -485.279} C_VEL
LIN {X 0,Y 608.466,Z 262.319,A -85,B 0,C 180,E1 -488.24,E2 -488.24} C_VEL
LIN {X 0,Y 608.412,Z 262.317,A -85,B 0,C 180,E1 -491.179,E2 -491.179} C_VEL
LIN {X 0,Y 608.47,Z 262.318,A -85,B 0,C 180,E1 -493.869,E2 -493.869} C_VEL
LIN {X 0,Y 608.429,Z 262.316,A -85,B 0,C 180,E1 -496.694,E2 -496.694} C_VEL
LIN {X 0,Y 608.403,Z 262.319,A -85,B 0,C 180,E1 -498.819,E2 -498.819} C_VEL
LIN {X 0,Y 608.46,Z 262.318,A -85,B 0,C 180,E1 -501.759,E2 -501.759} C_VEL
LIN {X 0,Y 608.406,Z 262.318,A -85,B 0,C 180,E1 -504.719,E2 -504.719} C_VEL
LIN {X 0,Y 608.454,Z 262.316,A -85,B 0,C 180,E1 -507.477,E2 -507.477} C_VEL
LIN {X 0,Y 608.442,Z 262.318,A -85,B 0,C 180,E1 -510.218,E2 -510.218} C_VEL
LIN {X 0,Y 608.409,Z 262.318,A -85,B 0,C 180,E1 -512.804,E2 -512.804} C_VEL
LIN {X 0,Y 608.435,Z 262.319,A -85,B 0,C 180,E1 -515.427,E2 -515.427} C_VEL
LIN {X 0,Y 608.432,Z 262.317,A -85,B 0,C 180,E1 -518.306,E2 -518.306} C_VEL
LIN {X 0,Y 608.409,Z 262.319,A -85,B 0,C 180,E1 -520.427,E2 -520.427} C_VEL
LIN {X 0,Y 608.472,Z 262.316,A -85,B 0,C 180,E1 -523.466,E2 -523.466} C_VEL
LIN {X 0,Y 608.424,Z 262.321,A -85,B 0,C 180,E1 -525.996,E2 -525.996} C_VEL
LIN {X 0,Y 608.427,Z 262.32,A -85,B 0,C 180,E1 -527.999,E2 -527.999} C_VEL
LIN {X 0,Y 608.411,Z 262.317,A -85,B 0,C 180,E1 -530.692,E2 -530.692} C_VEL
LIN {X 0,Y 608.471,Z 262.316,A -85,B 0,C 180,E1 -533.366,E2 -533.366} C_VEL
LIN {X 0,Y 608.408,Z 262.321,A -85,B 0,C 180,E1 -536.025,E2 -536.025} C_VEL
LIN {X 0,Y 608.41,Z 262.321,A -85,B 0,C 180,E1 -538.013,E2 -538.013} C_VEL
LIN {X 0,Y 608.431,Z 262.318,A -85,B 0,C 180,E1 -539.999,E2 -539.999} C_VEL
LIN {X 0,Y 608.411,Z 262.318,A -85,B 0,C 180,E1 -542.647,E2 -542.647} C_VEL
LIN {X 0,Y 608.441,Z 262.321,A -85,B 0,C 180,E1 -545.301,E2 -545.301} C_VEL
LIN {X 0,Y 608.401,Z 262.321,A -85,B 0,C 180,E1 -547.967,E2 -547.967} C_VEL
LIN {X 0,Y 608.433,Z 262.321,A -85,B 0,C 180,E1 -549.404,E2 -549.404} C_VEL
LIN {X 0,Y 607.738,Z 262.404,A -85,B 0,C 180,E1 -549.956,E2 -549.956} C_VEL
LIN {X 0,Y 604.884,Z 262.759,A -85,B 0,C 180,E1 -550.853,E2 -550.853} C_VEL
LIN {X 0,Y 602.484,Z 263.064,A -85,B 0,C 180,E1 -551.574,E2 -551.574} C_VEL
LIN {X 0,Y 601.445,Z 263.187,A -85,B 0,C 180,E1 -552.131,E2 -552.131} C_VEL
LIN {X 0,Y 601.355,Z 263.196,A -85,B 0,C 180,E1 -552.319,E2 -552.319} C_VEL
LIN {X 0,Y 601.369,Z 263.197,A -85,B 0,C 180,E1 -554.897,E2 -554.897} C_VEL
LIN {X 0,Y 601.367,Z 263.199,A -85,B 0,C 180,E1 -557.688,E2 -557.688} C_VEL
LIN {X 0,Y 601.371,Z 263.197,A -85,B 0,C 180,E1 -559.809,E2 -559.809} C_VEL
LIN {X 0,Y 601.386,Z 263.194,A -85,B 0,C 180,E1 -562.682,E2 -562.682} C_VEL
LIN {X 0,Y 601.408,Z 263.193,A -85,B 0,C 180,E1 -565.617,E2 -565.617} C_VEL
LIN {X 0,Y 601.348,Z 263.198,A -85,B 0,C 180,E1 -567.869,E2 -567.869} C_VEL
LIN {X 0,Y 601.357,Z 263.196,A -85,B 0,C 180,E1 -570.166,E2 -570.166} C_VEL
LIN {X 0,Y 601.38,Z 263.194,A -85,B 0,C 180,E1 -572.517,E2 -572.517} C_VEL
LIN {X 0,Y 601.367,Z 263.205,A -85,B 0,C 180,E1 -575.109,E2 -575.109} C_VEL
LIN {X 0,Y 601.418,Z 263.194,A -85,B 0,C 180,E1 -577.418,E2 -577.418} C_VEL
LIN {X 0,Y 601.37,Z 263.195,A -85,B 0,C 180,E1 -579.996,E2 -579.996} C_VEL
LIN {X 0,Y 601.369,Z 263.199,A -85,B 0,C 180,E1 -582.672,E2 -582.672} C_VEL
LIN {X 0,Y 601.38,Z 263.196,A -85,B 0,C 180,E1 -585.479,E2 -585.479} C_VEL
LIN {X 0,Y 601.395,Z 263.193,A -85,B 0,C 180,E1 -588.407,E2 -588.407} C_VEL
LIN {X 0,Y 601.393,Z 263.201,A -85,B 0,C 180,E1 -590.873,E2 -590.873} C_VEL
LIN {X 0,Y 601.393,Z 263.195,A -85,B 0,C 180,E1 -593.417,E2 -593.417} C_VEL
LIN {X 0,Y 601.397,Z 263.191,A -85,B 0,C 180,E1 -596.066,E2 -596.066} C_VEL
LIN {X 0,Y 601.42,Z 263.193,A -85,B 0,C 180,E1 -598.541,E2 -598.541} C_VEL
LIN {X 0,Y 601.409,Z 263.192,A -85,B 0,C 180,E1 -601.372,E2 -601.372} C_VEL
LIN {X 0,Y 601.379,Z 263.194,A -85,B 0,C 180,E1 -603.635,E2 -603.635} C_VEL
LIN {X 0,Y 601.395,Z 263.198,A -85,B 0,C 180,E1 -606.589,E2 -606.589} C_VEL
LIN {X 0,Y 601.404,Z 263.191,A -85,B 0,C 180,E1 -609.477,E2 -609.477} C_VEL
LIN {X 0,Y 601.377,Z 263.197,A -85,B 0,C 180,E1 -612.311,E2 -612.311} C_VEL
LIN {X 0,Y 601.413,Z 263.194,A -85,B 0,C 180,E1 -615.103,E2 -615.103} C_VEL
LIN {X 0,Y 601.387,Z 263.193,A -85,B 0,C 180,E1 -617.857,E2 -617.857} C_VEL
LIN {X 0,Y 601.401,Z 263.191,A -85,B 0,C 180,E1 -619.904,E2 -619.904} C_VEL
LIN {X 0,Y 601.441,Z 263.196,A -85,B 0,C 180,E1 -622.615,E2 -622.615} C_VEL
LIN {X 0,Y 601.4,Z 263.192,A -85,B 0,C 180,E1 -625.308,E2 -625.308} C_VEL
LIN {X 0,Y 601.391,Z 263.194,A -85,B 0,C 180,E1 -627.991,E2 -627.991} C_VEL
LIN {X 0,Y 601.451,Z 263.194,A -85,B 0,C 180,E1 -630.669,E2 -630.669} C_VEL
LIN {X 0,Y 601.409,Z 263.191,A -85,B 0,C 180,E1 -633.349,E2 -633.349} C_VEL
LIN {X 0,Y 601.385,Z 263.197,A -85,B 0,C 180,E1 -636.037,E2 -636.037} C_VEL
LIN {X 0,Y 601.415,Z 263.31,A -85,B 0,C 180,E1 -637.448,E2 -637.448} C_VEL
LIN {X 0,Y 601.679,Z 269.042,A -85,B 0,C 180,E1 -638.226,E2 -638.226} C_VEL
LIN {X 0,Y 601.609,Z 290.886,A -85,B 0,C 180,E1 -641.113,E2 -641.113} C_VEL
LIN {X 0,Y 601.577,Z 292.868,A -85,B 0,C 180,E1 -641.371,E2 -641.371} C_VEL
LIN {X 0,Y 601.993,Z 297.201,A -85,B 0,C 180,E1 -641.447,E2 -641.447} C_VEL
LIN {X 0,Y 601.852,Z 458.476,A -85,B 0,C 180,E1 -643.441,E2 -643.441} C_VEL
LIN {X 0,Y 601.841,Z 474.233,A -85,B 0,C 180,E1 -643.784,E2 -643.784} C_VEL
LIN {X 0,Y 601.766,Z 489.806,A -85,B 0,C 180,E1 -644.274,E2 -644.274} C_VEL
LIN {X 0,Y 601.706,Z 504.505,A -85,B 0,C 180,E1 -644.889,E2 -644.889} C_VEL
LIN {X 0,Y 601.651,Z 517.742,A -85,B 0,C 180,E1 -645.584,E2 -645.584} C_VEL
LIN {X 0,Y 601.589,Z 530.77,A -85,B 0,C 180,E1 -646.417,E2 -646.417} C_VEL
LIN {X 0,Y 601.509,Z 543.746,A -85,B 0,C 180,E1 -647.421,E2 -647.421} C_VEL
LIN {X 0,Y 601.489,Z 555.304,A -85,B 0,C 180,E1 -648.499,E2 -648.499} C_VEL
LIN {X 0,Y 601.418,Z 565.472,A -85,B 0,C 180,E1 -649.63,E2 -649.63} C_VEL
LIN {X 0,Y 601.407,Z 574.292,A -85,B 0,C 180,E1 -650.798,E2 -650.798} C_VEL
LIN {X 0,Y 601.374,Z 581.615,A -85,B 0,C 180,E1 -651.96,E2 -651.96} C_VEL
LIN {X 0,Y 601.353,Z 587.337,A -85,B 0,C 180,E1 -653.048,E2 -653.048} C_VEL
LIN {X 0,Y 601.341,Z 592.682,A -85,B 0,C 180,E1 -654.277,E2 -654.277} C_VEL
LIN {X 0,Y 601.33,Z 597.22,A -85,B 0,C 180,E1 -655.621,E2 -655.621} C_VEL
LIN {X 0,Y 601.326,Z 600.772,A -85,B 0,C 180,E1 -657.116,E2 -657.116} C_VEL
LIN {X 0,Y 601.325,Z 602.86,A -85,B 0,C 180,E1 -658.631,E2 -658.631} C_VEL
LIN {X 0,Y 601.329,Z 603.477,A -85,B 0,C 180,E1 -660.168,E2 -660.168} C_VEL
LIN {X 0,Y 601.326,Z 602.569,A -85,B 0,C 180,E1 -661.73,E2 -661.73} C_VEL
LIN {X 0,Y 601.321,Z 601.218,A -85,B 0,C 180,E1 -662.704,E2 -662.704} C_VEL
LIN {X 0,Y 601.335,Z 598.138,A -85,B 0,C 180,E1 -664.123,E2 -664.123} C_VEL
LIN {X 0,Y 601.343,Z 594.175,A -85,B 0,C 180,E1 -665.407,E2 -665.407} C_VEL
LIN {X 0,Y 601.374,Z 589.492,A -85,B 0,C 180,E1 -666.584,E2 -666.584} C_VEL
LIN {X 0,Y 601.357,Z 583.199,A -85,B 0,C 180,E1 -667.846,E2 -667.846} C_VEL
LIN {X 0,Y 601.414,Z 575.395,A -85,B 0,C 180,E1 -669.125,E2 -669.125} C_VEL
LIN {X 0,Y 601.419,Z 567.501,A -85,B 0,C 180,E1 -670.206,E2 -670.206} C_VEL
LIN {X 0,Y 601.45,Z 557.943,A -85,B 0,C 180,E1 -671.314,E2 -671.314} C_VEL
LIN {X 0,Y 601.49,Z 546.697,A -85,B 0,C 180,E1 -672.409,E2 -672.409} C_VEL
LIN {X 0,Y 601.56,Z 535.284,A -85,B 0,C 180,E1 -673.342,E2 -673.342} C_VEL
LIN {X 0,Y 601.615,Z 521.74,A -85,B 0,C 180,E1 -674.264,E2 -674.264} C_VEL
LIN {X 0,Y 601.698,Z 507.66,A -85,B 0,C 180,E1 -675.045,E2 -675.045} C_VEL
LIN {X 0,Y 601.764,Z 493.764,A -85,B 0,C 180,E1 -675.663,E2 -675.663} C_VEL
LIN {X 0,Y 601.831,Z 478.722,A -85,B 0,C 180,E1 -676.179,E2 -676.179} C_VEL
LIN {X 0,Y 601.87,Z 463.63,A -85,B 0,C 180,E1 -676.552,E2 -676.552} C_VEL
LIN {X 0,Y 601.886,Z 446.598,A -85,B 0,C 180,E1 -676.814,E2 -676.814} C_VEL
LIN {X 0,Y 601.953,Z 294.771,A -85,B 0,C 180,E1 -678.674,E2 -678.674} C_VEL
LIN {X 0,Y 601.566,Z 292.809,A -85,B 0,C 180,E1 -678.727,E2 -678.727} C_VEL
LIN {X 0,Y 601.657,Z 271.775,A -85,B 0,C 180,E1 -681.5,E2 -681.5} C_VEL
LIN {X 0,Y 601.449,Z 263.39,A -85,B 0,C 180,E1 -682.63,E2 -682.63} C_VEL
LIN {X 0,Y 601.427,Z 263.191,A -85,B 0,C 180,E1 -685.071,E2 -685.071} C_VEL
LIN {X 0,Y 601.431,Z 263.198,A -85,B 0,C 180,E1 -687.486,E2 -687.486} C_VEL
LIN {X 0,Y 601.43,Z 263.192,A -85,B 0,C 180,E1 -689.849,E2 -689.849} C_VEL
LIN {X 0,Y 601.408,Z 263.191,A -85,B 0,C 180,E1 -692.636,E2 -692.636} C_VEL
LIN {X 0,Y 601.394,Z 263.198,A -85,B 0,C 180,E1 -695.123,E2 -695.123} C_VEL
LIN {X 0,Y 601.4,Z 263.201,A -85,B 0,C 180,E1 -697.395,E2 -697.395} C_VEL
LIN {X 0,Y 601.395,Z 263.192,A -85,B 0,C 180,E1 -700.192,E2 -700.192} C_VEL
LIN {X 0,Y 601.424,Z 263.195,A -85,B 0,C 180,E1 -703.015,E2 -703.015} C_VEL
LIN {X 0,Y 601.404,Z 263.191,A -85,B 0,C 180,E1 -705.909,E2 -705.909} C_VEL
LIN {X 0,Y 601.425,Z 263.19,A -85,B 0,C 180,E1 -708.543,E2 -708.543} C_VEL
LIN {X 0,Y 601.398,Z 263.199,A -85,B 0,C 180,E1 -711.263,E2 -711.263} C_VEL
LIN {X 0,Y 601.415,Z 263.194,A -85,B 0,C 180,E1 -713.346,E2 -713.346} C_VEL
LIN {X 0,Y 601.377,Z 263.194,A -85,B 0,C 180,E1 -715.98,E2 -715.98} C_VEL
LIN {X 0,Y 601.429,Z 263.193,A -85,B 0,C 180,E1 -718.662,E2 -718.662} C_VEL
LIN {X 0,Y 601.396,Z 263.195,A -85,B 0,C 180,E1 -721.34,E2 -721.34} C_VEL
LIN {X 0,Y 601.399,Z 263.194,A -85,B 0,C 180,E1 -723.351,E2 -723.351} C_VEL
LIN {X 0,Y 601.397,Z 263.194,A -85,B 0,C 180,E1 -725.365,E2 -725.365} C_VEL
LIN {X 0,Y 601.383,Z 263.195,A -85,B 0,C 180,E1 -727.387,E2 -727.387} C_VEL
LIN {X 0,Y 601.381,Z 263.195,A -85,B 0,C 180,E1 -729.417,E2 -729.417} C_VEL
LIN {X 0,Y 601.391,Z 263.193,A -85,B 0,C 180,E1 -731.46,E2 -731.46} C_VEL
LIN {X 0,Y 601.4,Z 263.194,A -85,B 0,C 180,E1 -734.207,E2 -734.207} C_VEL
LIN {X 0,Y 601.413,Z 263.194,A -85,B 0,C 180,E1 -736.987,E2 -736.987} C_VEL
LIN {X 0,Y 601.373,Z 263.195,A -85,B 0,C 180,E1 -739.811,E2 -739.811} C_VEL
LIN {X 0,Y 601.384,Z 263.195,A -85,B 0,C 180,E1 -741.961,E2 -741.961} C_VEL
LIN {X 0,Y 601.412,Z 263.196,A -85,B 0,C 180,E1 -744.291,E2 -744.291} C_VEL
LIN {X 0,Y 601.37,Z 263.196,A -85,B 0,C 180,E1 -747.116,E2 -747.116} C_VEL
LIN {X 0,Y 601.363,Z 263.195,A -85,B 0,C 180,E1 -749.397,E2 -749.397} C_VEL
LIN {X 0,Y 601.421,Z 263.196,A -85,B 0,C 180,E1 -752.517,E2 -752.517} C_VEL
LIN {X 0,Y 601.346,Z 263.198,A -85,B 0,C 180,E1 -755.107,E2 -755.107} C_VEL
LIN {X 0,Y 601.373,Z 263.195,A -85,B 0,C 180,E1 -757.424,E2 -757.424} C_VEL
LIN {X 0,Y 601.384,Z 263.2,A -85,B 0,C 180,E1 -759.998,E2 -759.998} C_VEL
LIN {X 0,Y 601.37,Z 263.197,A -85,B 0,C 180,E1 -762.674,E2 -762.674} C_VEL
LIN {X 0,Y 601.392,Z 263.194,A -85,B 0,C 180,E1 -765.48,E2 -765.48} C_VEL
LIN {X 0,Y 601.401,Z 263.195,A -85,B 0,C 180,E1 -768.41,E2 -768.41} C_VEL
LIN {X 0,Y 601.378,Z 263.194,A -85,B 0,C 180,E1 -770.872,E2 -770.872} C_VEL
LIN {X 0,Y 601.385,Z 263.199,A -85,B 0,C 180,E1 -773.742,E2 -773.742} C_VEL
LIN {X 0,Y 601.402,Z 263.192,A -85,B 0,C 180,E1 -776.686,E2 -776.686} C_VEL
LIN {X 0,Y 601.397,Z 263.192,A -85,B 0,C 180,E1 -779.058,E2 -779.058} C_VEL
LIN {X 0,Y 601.406,Z 263.194,A -85,B 0,C 180,E1 -781.373,E2 -781.373} C_VEL
LIN {X 0,Y 601.403,Z 263.196,A -85,B 0,C 180,E1 -784.382,E2 -784.382} C_VEL
LIN {X 0,Y 601.407,Z 263.235,A -85,B 0,C 180,E1 -784.521,E2 -784.521} C_VEL
LIN {X 0,Y 601.843,Z 266.746,A -85,B 0,C 180,E1 -784.957,E2 -784.957} C_VEL
LIN {X 0,Y 601.769,Z 289.079,A -85,B 0,C 180,E1 -787.569,E2 -787.569} C_VEL
LIN {X 0,Y 601.686,Z 313.565,A -85,B 0,C 180,E1 -790.379,E2 -790.379} C_VEL
LIN {X 0,Y 601.628,Z 321.875,A -85,B 0,C 180,E1 -791.32,E2 -791.32} C_VEL
LIN {X 0,Y 602.027,Z 326.078,A -85,B 0,C 180,E1 -791.389,E2 -791.389} C_VEL
LIN {X 0,Y 601.878,Z 488.512,A -85,B 0,C 180,E1 -793.397,E2 -793.397} C_VEL
LIN {X 0,Y 601.815,Z 504.509,A -85,B 0,C 180,E1 -793.746,E2 -793.746} C_VEL
LIN {X 0,Y 601.767,Z 519.065,A -85,B 0,C 180,E1 -794.202,E2 -794.202} C_VEL
LIN {X 0,Y 601.72,Z 532.774,A -85,B 0,C 180,E1 -794.765,E2 -794.765} C_VEL
LIN {X 0,Y 601.662,Z 546.244,A -85,B 0,C 180,E1 -795.456,E2 -795.456} C_VEL
LIN {X 0,Y 601.617,Z 559.456,A -85,B 0,C 180,E1 -796.284,E2 -796.284} C_VEL
LIN {X 0,Y 601.532,Z 571.291,A -85,B 0,C 180,E1 -797.175,E2 -797.175} C_VEL
LIN {X 0,Y 601.488,Z 582.754,A -85,B 0,C 180,E1 -798.202,E2 -798.202} C_VEL
LIN {X 0,Y 601.431,Z 592.393,A -85,B 0,C 180,E1 -799.225,E2 -799.225} C_VEL
LIN {X 0,Y 601.428,Z 601.858,A -85,B 0,C 180,E1 -800.415,E2 -800.415} C_VEL
LIN {X 0,Y 601.368,Z 609.733,A -85,B 0,C 180,E1 -801.6,E2 -801.6} C_VEL
LIN {X 0,Y 601.368,Z 617.09,A -85,B 0,C 180,E1 -802.952,E2 -802.952} C_VEL
LIN {X 0,Y 601.371,Z 622.925,A -85,B 0,C 180,E1 -804.299,E2 -804.299} C_VEL
LIN {X 0,Y 601.33,Z 626.384,A -85,B 0,C 180,E1 -805.308,E2 -805.308} C_VEL
LIN {X 0,Y 601.337,Z 629.887,A -85,B 0,C 180,E1 -806.65,E2 -806.65} C_VEL
LIN {X 0,Y 601.341,Z 632.192,A -85,B 0,C 180,E1 -807.991,E2 -807.991} C_VEL
LIN {X 0,Y 601.337,Z 633.35,A -85,B 0,C 180,E1 -809.331,E2 -809.331} C_VEL
LIN {X 0,Y 601.337,Z 633.35,A -85,B 0,C 180,E1 -810.67,E2 -810.67} C_VEL
LIN {X 0,Y 601.341,Z 632.191,A -85,B 0,C 180,E1 -812.01,E2 -812.01} C_VEL
LIN {X 0,Y 601.337,Z 629.885,A -85,B 0,C 180,E1 -813.35,E2 -813.35} C_VEL
LIN {X 0,Y 601.33,Z 626.383,A -85,B 0,C 180,E1 -814.693,E2 -814.693} C_VEL
LIN {X 0,Y 601.352,Z 621.607,A -85,B 0,C 180,E1 -816.038,E2 -816.038} C_VEL
LIN {X 0,Y 601.366,Z 615.425,A -85,B 0,C 180,E1 -817.386,E2 -817.386} C_VEL
LIN {X 0,Y 601.387,Z 607.652,A -85,B 0,C 180,E1 -818.738,E2 -818.738} C_VEL
LIN {X 0,Y 601.427,Z 599.37,A -85,B 0,C 180,E1 -819.925,E2 -819.925} C_VEL
LIN {X 0,Y 601.461,Z 588.932,A -85,B 0,C 180,E1 -821.165,E2 -821.165} C_VEL
LIN {X 0,Y 601.514,Z 579.192,A -85,B 0,C 180,E1 -822.14,E2 -822.14} C_VEL
LIN {X 0,Y 601.57,Z 567.016,A -85,B 0,C 180,E1 -823.168,E2 -823.168} C_VEL
LIN {X 0,Y 601.607,Z 555.078,A -85,B 0,C 180,E1 -824.011,E2 -824.011} C_VEL
LIN {X 0,Y 601.669,Z 541.527,A -85,B 0,C 180,E1 -824.804,E2 -824.804} C_VEL
LIN {X 0,Y 601.765,Z 526.843,A -85,B 0,C 180,E1 -825.495,E2 -825.495} C_VEL
LIN {X 0,Y 601.788,Z 512.62,A -85,B 0,C 180,E1 -826.016,E2 -826.016} C_VEL
LIN {X 0,Y 601.86,Z 497.674,A -85,B 0,C 180,E1 -826.42,E2 -826.42} C_VEL
LIN {X 0,Y 601.87,Z 482.689,A -85,B 0,C 180,E1 -826.69,E2 -826.69} C_VEL
LIN {X 0,Y 601.904,Z 323.495,A -85,B 0,C 180,E1 -828.647,E2 -828.647} C_VEL
LIN {X 0,Y 601.628,Z 321.75,A -85,B 0,C 180,E1 -828.694,E2 -828.694} C_VEL
LIN {X 0,Y 601.75,Z 296.393,A -85,B 0,C 180,E1 -831.586,E2 -831.586} C_VEL
LIN {X 0,Y 601.876,Z 272.31,A -85,B 0,C 180,E1 -834.385,E2 -834.385} C_VEL
LIN {X 0,Y 601.82,Z 265.181,A -85,B 0,C 180,E1 -835.229,E2 -835.229} C_VEL
LIN {X 0,Y 601.415,Z 263.195,A -85,B 0,C 180,E1 -835.502,E2 -835.502} C_VEL
LIN {X 0,Y 601.409,Z 263.194,A -85,B 0,C 180,E1 -838.628,E2 -838.628} C_VEL
LIN {X 0,Y 601.399,Z 263.192,A -85,B 0,C 180,E1 -840.943,E2 -840.943} C_VEL
LIN {X 0,Y 601.405,Z 263.191,A -85,B 0,C 180,E1 -843.314,E2 -843.314} C_VEL
LIN {X 0,Y 601.39,Z 263.201,A -85,B 0,C 180,E1 -846.259,E2 -846.259} C_VEL
LIN {X 0,Y 601.384,Z 263.193,A -85,B 0,C 180,E1 -849.128,E2 -849.128} C_VEL
LIN {X 0,Y 601.418,Z 263.194,A -85,B 0,C 180,E1 -851.765,E2 -851.765} C_VEL
LIN {X 0,Y 601.395,Z 263.194,A -85,B 0,C 180,E1 -854.532,E2 -854.532} C_VEL
LIN {X 0,Y 601.384,Z 263.195,A -85,B 0,C 180,E1 -857.411,E2 -857.411} C_VEL
LIN {X 0,Y 601.392,Z 263.202,A -85,B 0,C 180,E1 -860.003,E2 -860.003} C_VEL
LIN {X 0,Y 601.387,Z 263.194,A -85,B 0,C 180,E1 -862.623,E2 -862.623} C_VEL
LIN {X 0,Y 601.372,Z 263.194,A -85,B 0,C 180,E1 -865.065,E2 -865.065} C_VEL
LIN {X 0,Y 601.422,Z 263.192,A -85,B 0,C 180,E1 -867.483,E2 -867.483} C_VEL
LIN {X 0,Y 601.402,Z 263.201,A -85,B 0,C 180,E1 -869.854,E2 -869.854} C_VEL
LIN {X 0,Y 601.386,Z 263.198,A -85,B 0,C 180,E1 -872.13,E2 -872.13} C_VEL
LIN {X 0,Y 601.377,Z 263.196,A -85,B 0,C 180,E1 -874.379,E2 -874.379} C_VEL
LIN {X 0,Y 601.364,Z 263.196,A -85,B 0,C 180,E1 -876.587,E2 -876.587} C_VEL
LIN {X 0,Y 601.417,Z 263.194,A -85,B 0,C 180,E1 -879.477,E2 -879.477} C_VEL
LIN {X 0,Y 601.359,Z 263.198,A -85,B 0,C 180,E1 -882.31,E2 -882.31} C_VEL
LIN {X 0,Y 601.37,Z 263.195,A -85,B 0,C 180,E1 -884.407,E2 -884.407} C_VEL
LIN {X 0,Y 601.391,Z 263.194,A -85,B 0,C 180,E1 -887.17,E2 -887.17} C_VEL
LIN {X 0,Y 601.382,Z 263.199,A -85,B 0,C 180,E1 -889.903,E2 -889.903} C_VEL
LIN {X 0,Y 601.354,Z 263.197,A -85,B 0,C 180,E1 -892.613,E2 -892.613} C_VEL
LIN {X 0,Y 601.409,Z 263.195,A -85,B 0,C 180,E1 -895.307,E2 -895.307} C_VEL
LIN {X 0,Y 601.384,Z 263.196,A -85,B 0,C 180,E1 -897.99,E2 -897.99} C_VEL
LIN {X 0,Y 601.403,Z 263.194,A -85,B 0,C 180,E1 -899.999,E2 -899.999} C_VEL
LIN {X 0,Y 601.383,Z 263.193,A -85,B 0,C 180,E1 -902.678,E2 -902.678} C_VEL
LIN {X 0,Y 601.403,Z 263.199,A -85,B 0,C 180,E1 -905.363,E2 -905.363} C_VEL
LIN {X 0,Y 601.375,Z 263.195,A -85,B 0,C 180,E1 -908.06,E2 -908.06} C_VEL
LIN {X 0,Y 601.362,Z 263.197,A -85,B 0,C 180,E1 -910.776,E2 -910.776} C_VEL
LIN {X 0,Y 601.355,Z 263.196,A -85,B 0,C 180,E1 -912.319,E2 -912.319} C_VEL
LIN {X 0,Y 600.678,Z 263.284,A -85,B 0,C 180,E1 -912.879,E2 -912.879} C_VEL
LIN {X 0,Y 597.832,Z 263.64,A -85,B 0,C 180,E1 -913.786,E2 -913.786} C_VEL
LIN {X 0,Y 595.433,Z 263.94,A -85,B 0,C 180,E1 -914.517,E2 -914.517} C_VEL
LIN {X 0,Y 594.401,Z 264.068,A -85,B 0,C 180,E1 -915.08,E2 -915.08} C_VEL
LIN {X 0,Y 594.316,Z 264.076,A -85,B 0,C 180,E1 -915.271,E2 -915.271} C_VEL
LIN {X 0,Y 594.312,Z 264.075,A -85,B 0,C 180,E1 -917.905,E2 -917.905} C_VEL
LIN {X 0,Y 594.361,Z 264.07,A -85,B 0,C 180,E1 -920.775,E2 -920.775} C_VEL
LIN {X 0,Y 594.33,Z 264.075,A -85,B 0,C 180,E1 -923.705,E2 -923.705} C_VEL
LIN {X 0,Y 594.333,Z 264.07,A -85,B 0,C 180,E1 -926.014,E2 -926.014} C_VEL
LIN {X 0,Y 594.306,Z 264.073,A -85,B 0,C 180,E1 -928.229,E2 -928.229} C_VEL
LIN {X 0,Y 594.345,Z 264.071,A -85,B 0,C 180,E1 -930.56,E2 -930.56} C_VEL
LIN {X 0,Y 594.355,Z 264.075,A -85,B 0,C 180,E1 -932.95,E2 -932.95} C_VEL
LIN {X 0,Y 594.309,Z 264.079,A -85,B 0,C 180,E1 -935.41,E2 -935.41} C_VEL
LIN {X 0,Y 594.352,Z 264.068,A -85,B 0,C 180,E1 -937.941,E2 -937.941} C_VEL
LIN {X 0,Y 594.36,Z 264.074,A -85,B 0,C 180,E1 -940.821,E2 -940.821} C_VEL
LIN {X 0,Y 594.342,Z 264.07,A -85,B 0,C 180,E1 -943.838,E2 -943.838} C_VEL
LIN {X 0,Y 594.332,Z 264.075,A -85,B 0,C 180,E1 -946.698,E2 -946.698} C_VEL
LIN {X 0,Y 594.343,Z 264.074,A -85,B 0,C 180,E1 -949.432,E2 -949.432} C_VEL
LIN {X 0,Y 594.367,Z 264.068,A -85,B 0,C 180,E1 -952.391,E2 -952.391} C_VEL
LIN {X 0,Y 594.381,Z 264.068,A -85,B 0,C 180,E1 -955.421,E2 -955.421} C_VEL
LIN {X 0,Y 594.367,Z 264.069,A -85,B 0,C 180,E1 -958.355,E2 -958.355} C_VEL
LIN {X 0,Y 594.362,Z 264.075,A -85,B 0,C 180,E1 -961.042,E2 -961.042} C_VEL
LIN {X 0,Y 594.37,Z 264.07,A -85,B 0,C 180,E1 -963.3,E2 -963.3} C_VEL
LIN {X 0,Y 594.359,Z 264.07,A -85,B 0,C 180,E1 -966.295,E2 -966.295} C_VEL
LIN {X 0,Y 594.384,Z 264.068,A -85,B 0,C 180,E1 -969.224,E2 -969.224} C_VEL
LIN {X 0,Y 594.327,Z 264.074,A -85,B 0,C 180,E1 -972.094,E2 -972.094} C_VEL
LIN {X 0,Y 594.345,Z 264.072,A -85,B 0,C 180,E1 -974.219,E2 -974.219} C_VEL
LIN {X 0,Y 594.351,Z 264.074,A -85,B 0,C 180,E1 -977.017,E2 -977.017} C_VEL
LIN {X 0,Y 594.386,Z 264.068,A -85,B 0,C 180,E1 -979.095,E2 -979.095} C_VEL
LIN {X 0,Y 594.358,Z 264.069,A -85,B 0,C 180,E1 -981.842,E2 -981.842} C_VEL
LIN {X 0,Y 594.387,Z 264.075,A -85,B 0,C 180,E1 -984.572,E2 -984.572} C_VEL
LIN {X 0,Y 594.387,Z 264.066,A -85,B 0,C 180,E1 -987.289,E2 -987.289} C_VEL
LIN {X 0,Y 594.381,Z 264.068,A -85,B 0,C 180,E1 -990,E2 -990} C_VEL
LIN {X 0,Y 594.409,Z 264.07,A -85,B 0,C 180,E1 -992.71,E2 -992.71} C_VEL
LIN {X 0,Y 594.371,Z 264.068,A -85,B 0,C 180,E1 -995.428,E2 -995.428} C_VEL
LIN {X 0,Y 594.406,Z 264.144,A -85,B 0,C 180,E1 -997.28,E2 -997.28} C_VEL
LIN {X 0,Y 594.757,Z 267.939,A -85,B 0,C 180,E1 -997.81,E2 -997.81} C_VEL
LIN {X 0,Y 594.658,Z 287.127,A -85,B 0,C 180,E1 -1000.383,E2 -1000.383} C_VEL
LIN {X 0,Y 594.642,Z 292.891,A -85,B 0,C 180,E1 -1001.148,E2 -1001.148} C_VEL
LIN {X 0,Y 595.268,Z 296.86,A -85,B 0,C 180,E1 -1001.225,E2 -1001.225} C_VEL
LIN {X 0,Y 595.073,Z 457.351,A -85,B 0,C 180,E1 -1003.227,E2 -1003.227} C_VEL
LIN {X 0,Y 595.031,Z 472.782,A -85,B 0,C 180,E1 -1003.554,E2 -1003.554} C_VEL
LIN {X 0,Y 594.952,Z 487.578,A -85,B 0,C 180,E1 -1004.008,E2 -1004.008} C_VEL
LIN {X 0,Y 594.827,Z 502.741,A -85,B 0,C 180,E1 -1004.627,E2 -1004.627} C_VEL
LIN {X 0,Y 594.734,Z 516.322,A -85,B 0,C 180,E1 -1005.331,E2 -1005.331} C_VEL
LIN {X 0,Y 594.633,Z 530.17,A -85,B 0,C 180,E1 -1006.213,E2 -1006.213} C_VEL
LIN {X 0,Y 594.552,Z 542.762,A -85,B 0,C 180,E1 -1007.188,E2 -1007.188} C_VEL
LIN {X 0,Y 594.462,Z 554.298,A -85,B 0,C 180,E1 -1008.257,E2 -1008.257} C_VEL
LIN {X 0,Y 594.395,Z 564.05,A -85,B 0,C 180,E1 -1009.333,E2 -1009.333} C_VEL
LIN {X 0,Y 594.362,Z 573.652,A -85,B 0,C 180,E1 -1010.595,E2 -1010.595} C_VEL
LIN {X 0,Y 594.304,Z 581.649,A -85,B 0,C 180,E1 -1011.869,E2 -1011.869} C_VEL
LIN {X 0,Y 594.289,Z 587.364,A -85,B 0,C 180,E1 -1012.969,E2 -1012.969} C_VEL
LIN {X 0,Y 594.26,Z 593.564,A -85,B 0,C 180,E1 -1014.451,E2 -1014.451} C_VEL
LIN {X 0,Y 594.224,Z 598.223,A -85,B 0,C 180,E1 -1015.95,E2 -1015.95} C_VEL
LIN {X 0,Y 594.245,Z 601.462,A -85,B 0,C 180,E1 -1017.505,E2 -1017.505} C_VEL
LIN {X 0,Y 594.237,Z 603.13,A -85,B 0,C 180,E1 -1019.005,E2 -1019.005} C_VEL
LIN {X 0,Y 594.219,Z 603.386,A -85,B 0,C 180,E1 -1020.568,E2 -1020.568} C_VEL
LIN {X 0,Y 594.229,Z 602.716,A -85,B 0,C 180,E1 -1021.623,E2 -1021.623} C_VEL
LIN {X 0,Y 594.232,Z 600.857,A -85,B 0,C 180,E1 -1022.958,E2 -1022.958} C_VEL
LIN {X 0,Y 594.255,Z 598.263,A -85,B 0,C 180,E1 -1024.124,E2 -1024.124} C_VEL
LIN {X 0,Y 594.259,Z 594.381,A -85,B 0,C 180,E1 -1025.414,E2 -1025.414} C_VEL
LIN {X 0,Y 594.284,Z 589.074,A -85,B 0,C 180,E1 -1026.757,E2 -1026.757} C_VEL
LIN {X 0,Y 594.315,Z 582.163,A -85,B 0,C 180,E1 -1028.132,E2 -1028.132} C_VEL
LIN {X 0,Y 594.36,Z 573.892,A -85,B 0,C 180,E1 -1029.461,E2 -1029.461} C_VEL
LIN {X 0,Y 594.411,Z 564.579,A -85,B 0,C 180,E1 -1030.694,E2 -1030.694} C_VEL
LIN {X 0,Y 594.468,Z 554.019,A -85,B 0,C 180,E1 -1031.86,E2 -1031.86} C_VEL
LIN {X 0,Y 594.533,Z 543.122,A -85,B 0,C 180,E1 -1032.872,E2 -1032.872} C_VEL
LIN {X 0,Y 594.645,Z 530.26,A -85,B 0,C 180,E1 -1033.87,E2 -1033.87} C_VEL
LIN {X 0,Y 594.726,Z 517.887,A -85,B 0,C 180,E1 -1034.669,E2 -1034.669} C_VEL
LIN {X 0,Y 594.829,Z 504.426,A -85,B 0,C 180,E1 -1035.384,E2 -1035.384} C_VEL
LIN {X 0,Y 594.918,Z 489.622,A -85,B 0,C 180,E1 -1036.009,E2 -1036.009} C_VEL
LIN {X 0,Y 595.013,Z 474.041,A -85,B 0,C 180,E1 -1036.503,E2 -1036.503} C_VEL
LIN {X 0,Y 595.084,Z 458.465,A -85,B 0,C 180,E1 -1036.843,E2 -1036.843} C_VEL
LIN {X 0,Y 595.215,Z 334.967,A -85,B 0,C 180,E1 -1038.392,E2 -1038.392} C_VEL
LIN {X 0,Y 595.197,Z 295.884,A -85,B 0,C 180,E1 -1038.88,E2 -1038.88} C_VEL
LIN {X 0,Y 594.645,Z 292.745,A -85,B 0,C 180,E1 -1038.961,E2 -1038.961} C_VEL
LIN {X 0,Y 594.775,Z 270.875,A -85,B 0,C 180,E1 -1041.883,E2 -1041.883} C_VEL
LIN {X 0,Y 594.447,Z 264.191,A -85,B 0,C 180,E1 -1042.802,E2 -1042.802} C_VEL
LIN {X 0,Y 594.373,Z 264.073,A -85,B 0,C 180,E1 -1045.86,E2 -1045.86} C_VEL
LIN {X 0,Y 594.377,Z 264.067,A -85,B 0,C 180,E1 -1048.652,E2 -1048.652} C_VEL
LIN {X 0,Y 594.375,Z 264.071,A -85,B 0,C 180,E1 -1051.041,E2 -1051.041} C_VEL
LIN {X 0,Y 594.375,Z 264.069,A -85,B 0,C 180,E1 -1053.976,E2 -1053.976} C_VEL
LIN {X 0,Y 594.377,Z 264.067,A -85,B 0,C 180,E1 -1056.297,E2 -1056.297} C_VEL
LIN {X 0,Y 594.396,Z 264.073,A -85,B 0,C 180,E1 -1059.226,E2 -1059.226} C_VEL
LIN {X 0,Y 594.367,Z 264.068,A -85,B 0,C 180,E1 -1062.097,E2 -1062.097} C_VEL
LIN {X 0,Y 594.355,Z 264.069,A -85,B 0,C 180,E1 -1064.22,E2 -1064.22} C_VEL
LIN {X 0,Y 594.359,Z 264.076,A -85,B 0,C 180,E1 -1067.018,E2 -1067.018} C_VEL
LIN {X 0,Y 594.374,Z 264.068,A -85,B 0,C 180,E1 -1069.785,E2 -1069.785} C_VEL
LIN {X 0,Y 594.407,Z 264.065,A -85,B 0,C 180,E1 -1072.528,E2 -1072.528} C_VEL
LIN {X 0,Y 594.373,Z 264.073,A -85,B 0,C 180,E1 -1075.253,E2 -1075.253} C_VEL
LIN {X 0,Y 594.368,Z 264.067,A -85,B 0,C 180,E1 -1077.968,E2 -1077.968} C_VEL
LIN {X 0,Y 594.423,Z 264.066,A -85,B 0,C 180,E1 -1080.679,E2 -1080.679} C_VEL
LIN {X 0,Y 594.35,Z 264.072,A -85,B 0,C 180,E1 -1083.391,E2 -1083.391} C_VEL
LIN {X 0,Y 594.361,Z 264.07,A -85,B 0,C 180,E1 -1085.429,E2 -1085.429} C_VEL
LIN {X 0,Y 594.35,Z 264.071,A -85,B 0,C 180,E1 -1088.159,E2 -1088.159} C_VEL
LIN {X 0,Y 594.386,Z 264.069,A -85,B 0,C 180,E1 -1091.079,E2 -1091.079} C_VEL
LIN {X 0,Y 594.363,Z 264.07,A -85,B 0,C 180,E1 -1094.169,E2 -1094.169} C_VEL
LIN {X 0,Y 594.367,Z 264.069,A -85,B 0,C 180,E1 -1097.195,E2 -1097.195} C_VEL
LIN {X 0,Y 594.352,Z 264.072,A -85,B 0,C 180,E1 -1100.055,E2 -1100.055} C_VEL
LIN {X 0,Y 594.336,Z 264.074,A -85,B 0,C 180,E1 -1102.969,E2 -1102.969} C_VEL
LIN {X 0,Y 594.31,Z 264.075,A -85,B 0,C 180,E1 -1105.197,E2 -1105.197} C_VEL
LIN {X 0,Y 594.332,Z 264.072,A -85,B 0,C 180,E1 -1107.52,E2 -1107.52} C_VEL
LIN {X 0,Y 594.336,Z 264.073,A -85,B 0,C 180,E1 -1109.779,E2 -1109.779} C_VEL
LIN {X 0,Y 594.35,Z 264.076,A -85,B 0,C 180,E1 -1112.149,E2 -1112.149} C_VEL
LIN {X 0,Y 594.34,Z 264.076,A -85,B 0,C 180,E1 -1114.583,E2 -1114.583} C_VEL
LIN {X 0,Y 594.342,Z 264.072,A -85,B 0,C 180,E1 -1117.605,E2 -1117.605} C_VEL
LIN {X 0,Y 594.331,Z 264.075,A -85,B 0,C 180,E1 -1119.771,E2 -1119.771} C_VEL
LIN {X 0,Y 594.341,Z 264.077,A -85,B 0,C 180,E1 -1122.378,E2 -1122.378} C_VEL
LIN {X 0,Y 594.33,Z 264.072,A -85,B 0,C 180,E1 -1125.195,E2 -1125.195} C_VEL
LIN {X 0,Y 594.365,Z 264.076,A -85,B 0,C 180,E1 -1128.154,E2 -1128.154} C_VEL
LIN {X 0,Y 594.358,Z 264.07,A -85,B 0,C 180,E1 -1131.299,E2 -1131.299} C_VEL
LIN {X 0,Y 594.34,Z 264.077,A -85,B 0,C 180,E1 -1133.756,E2 -1133.756} C_VEL
LIN {X 0,Y 594.366,Z 264.073,A -85,B 0,C 180,E1 -1136.239,E2 -1136.239} C_VEL
LIN {X 0,Y 594.357,Z 264.069,A -85,B 0,C 180,E1 -1138.65,E2 -1138.65} C_VEL
LIN {X 0,Y 594.371,Z 264.068,A -85,B 0,C 180,E1 -1141.045,E2 -1141.045} C_VEL
LIN {X 0,Y 594.38,Z 264.074,A -85,B 0,C 180,E1 -1144.245,E2 -1144.245} C_VEL
LIN {X 0,Y 594.432,Z 264.406,A -85,B 0,C 180,E1 -1144.342,E2 -1144.342} C_VEL
LIN {X 0,Y 595.046,Z 268.307,A -85,B 0,C 180,E1 -1144.838,E2 -1144.838} C_VEL
LIN {X 0,Y 594.908,Z 291.948,A -85,B 0,C 180,E1 -1147.633,E2 -1147.633} C_VEL
LIN {X 0,Y 594.76,Z 316.686,A -85,B 0,C 180,E1 -1150.5,E2 -1150.5} C_VEL
LIN {X 0,Y 594.7,Z 321.893,A -85,B 0,C 180,E1 -1151.096,E2 -1151.096} C_VEL
LIN {X 0,Y 595.313,Z 325.462,A -85,B 0,C 180,E1 -1151.164,E2 -1151.164} C_VEL
LIN {X 0,Y 595.084,Z 488.349,A -85,B 0,C 180,E1 -1153.199,E2 -1153.199} C_VEL
LIN {X 0,Y 595.019,Z 503.734,A -85,B 0,C 180,E1 -1153.533,E2 -1153.533} C_VEL
LIN {X 0,Y 594.933,Z 519.063,A -85,B 0,C 180,E1 -1154.015,E2 -1154.015} C_VEL
LIN {X 0,Y 594.857,Z 532.777,A -85,B 0,C 180,E1 -1154.584,E2 -1154.584} C_VEL
LIN {X 0,Y 594.737,Z 546.247,A -85,B 0,C 180,E1 -1155.282,E2 -1155.282} C_VEL
LIN {X 0,Y 594.68,Z 558.802,A -85,B 0,C 180,E1 -1156.076,E2 -1156.076} C_VEL
LIN {X 0,Y 594.56,Z 571.293,A -85,B 0,C 180,E1 -1157.022,E2 -1157.022} C_VEL
LIN {X 0,Y 594.465,Z 582.754,A -85,B 0,C 180,E1 -1158.06,E2 -1158.06} C_VEL
LIN {X 0,Y 594.389,Z 592.394,A -85,B 0,C 180,E1 -1159.095,E2 -1159.095} C_VEL
LIN {X 0,Y 594.366,Z 601.859,A -85,B 0,C 180,E1 -1160.3,E2 -1160.3} C_VEL
LIN {X 0,Y 594.311,Z 609.734,A -85,B 0,C 180,E1 -1161.5,E2 -1161.5} C_VEL
LIN {X 0,Y 594.292,Z 617.09,A -85,B 0,C 180,E1 -1162.868,E2 -1162.868} C_VEL
LIN {X 0,Y 594.296,Z 622.925,A -85,B 0,C 180,E1 -1164.231,E2 -1164.231} C_VEL
LIN {X 0,Y 594.232,Z 626.385,A -85,B 0,C 180,E1 -1165.251,E2 -1165.251} C_VEL
LIN {X 0,Y 594.256,Z 629.888,A -85,B 0,C 180,E1 -1166.61,E2 -1166.61} C_VEL
LIN {X 0,Y 594.24,Z 632.193,A -85,B 0,C 180,E1 -1167.967,E2 -1167.967} C_VEL
LIN {X 0,Y 594.237,Z 633.35,A -85,B 0,C 180,E1 -1169.323,E2 -1169.323} C_VEL
LIN {X 0,Y 594.237,Z 633.35,A -85,B 0,C 180,E1 -1170.678,E2 -1170.678} C_VEL
LIN {X 0,Y 594.24,Z 632.192,A -85,B 0,C 180,E1 -1172.034,E2 -1172.034} C_VEL
LIN {X 0,Y 594.256,Z 629.886,A -85,B 0,C 180,E1 -1173.39,E2 -1173.39} C_VEL
LIN {X 0,Y 594.232,Z 626.383,A -85,B 0,C 180,E1 -1174.749,E2 -1174.749} C_VEL
LIN {X 0,Y 594.275,Z 621.607,A -85,B 0,C 180,E1 -1176.11,E2 -1176.11} C_VEL
LIN {X 0,Y 594.287,Z 615.424,A -85,B 0,C 180,E1 -1177.475,E2 -1177.475} C_VEL
LIN {X 0,Y 594.331,Z 607.651,A -85,B 0,C 180,E1 -1178.843,E2 -1178.843} C_VEL
LIN {X 0,Y 594.387,Z 599.369,A -85,B 0,C 180,E1 -1180.044,E2 -1180.044} C_VEL
LIN {X 0,Y 594.434,Z 589.559,A -85,B 0,C 180,E1 -1181.231,E2 -1181.231} C_VEL
LIN {X 0,Y 594.531,Z 579.191,A -85,B 0,C 180,E1 -1182.285,E2 -1182.285} C_VEL
LIN {X 0,Y 594.581,Z 567.017,A -85,B 0,C 180,E1 -1183.326,E2 -1183.326} C_VEL
LIN {X 0,Y 594.695,Z 555.075,A -85,B 0,C 180,E1 -1184.178,E2 -1184.178} C_VEL
LIN {X 0,Y 594.782,Z 541.524,A -85,B 0,C 180,E1 -1184.98,E2 -1184.98} C_VEL
LIN {X 0,Y 594.906,Z 526.841,A -85,B 0,C 180,E1 -1185.678,E2 -1185.678} C_VEL
LIN {X 0,Y 594.967,Z 512.619,A -85,B 0,C 180,E1 -1186.205,E2 -1186.205} C_VEL
LIN {X 0,Y 595.052,Z 498.112,A -85,B 0,C 180,E1 -1186.603,E2 -1186.603} C_VEL
LIN {X 0,Y 595.07,Z 482.689,A -85,B 0,C 180,E1 -1186.886,E2 -1186.886} C_VEL
LIN {X 0,Y 595.217,Z 324.68,A -85,B 0,C 180,E1 -1188.849,E2 -1188.849} C_VEL
LIN {X 0,Y 594.71,Z 321.867,A -85,B 0,C 180,E1 -1188.907,E2 -1188.907} C_VEL
LIN {X 0,Y 594.885,Z 297.954,A -85,B 0,C 180,E1 -1191.665,E2 -1191.665} C_VEL
LIN {X 0,Y 595.045,Z 273.242,A -85,B 0,C 180,E1 -1194.572,E2 -1194.572} C_VEL
LIN {X 0,Y 594.955,Z 266.741,A -85,B 0,C 180,E1 -1195.354,E2 -1195.354} C_VEL
LIN {X 0,Y 594.37,Z 264.075,A -85,B 0,C 180,E1 -1195.709,E2 -1195.709} C_VEL
LIN {X 0,Y 594.362,Z 264.077,A -85,B 0,C 180,E1 -1198.227,E2 -1198.227} C_VEL
LIN {X 0,Y 594.375,Z 264.071,A -85,B 0,C 180,E1 -1200.56,E2 -1200.56} C_VEL
LIN {X 0,Y 594.371,Z 264.068,A -85,B 0,C 180,E1 -1202.95,E2 -1202.95} C_VEL
LIN {X 0,Y 594.32,Z 264.074,A -85,B 0,C 180,E1 -1205.411,E2 -1205.411} C_VEL
LIN {X 0,Y 594.372,Z 264.075,A -85,B 0,C 180,E1 -1207.941,E2 -1207.941} C_VEL
LIN {X 0,Y 594.355,Z 264.069,A -85,B 0,C 180,E1 -1210.819,E2 -1210.819} C_VEL
LIN {X 0,Y 594.338,Z 264.071,A -85,B 0,C 180,E1 -1213.301,E2 -1213.301} C_VEL
LIN {X 0,Y 594.341,Z 264.078,A -85,B 0,C 180,E1 -1216.162,E2 -1216.162} C_VEL
LIN {X 0,Y 594.36,Z 264.071,A -85,B 0,C 180,E1 -1218.534,E2 -1218.534} C_VEL
LIN {X 0,Y 594.361,Z 264.069,A -85,B 0,C 180,E1 -1221.297,E2 -1221.297} C_VEL
LIN {X 0,Y 594.341,Z 264.078,A -85,B 0,C 180,E1 -1223.754,E2 -1223.754} C_VEL
LIN {X 0,Y 594.356,Z 264.073,A -85,B 0,C 180,E1 -1226.237,E2 -1226.237} C_VEL
LIN {X 0,Y 594.352,Z 264.069,A -85,B 0,C 180,E1 -1228.648,E2 -1228.648} C_VEL
LIN {X 0,Y 594.369,Z 264.067,A -85,B 0,C 180,E1 -1231.043,E2 -1231.043} C_VEL
LIN {X 0,Y 594.333,Z 264.078,A -85,B 0,C 180,E1 -1234.053,E2 -1234.053} C_VEL
LIN {X 0,Y 594.357,Z 264.071,A -85,B 0,C 180,E1 -1236.294,E2 -1236.294} C_VEL
LIN {X 0,Y 594.389,Z 264.067,A -85,B 0,C 180,E1 -1239.223,E2 -1239.223} C_VEL
LIN {X 0,Y 594.317,Z 264.078,A -85,B 0,C 180,E1 -1242.093,E2 -1242.093} C_VEL
LIN {X 0,Y 594.332,Z 264.074,A -85,B 0,C 180,E1 -1244.217,E2 -1244.217} C_VEL
LIN {X 0,Y 594.339,Z 264.07,A -85,B 0,C 180,E1 -1246.319,E2 -1246.319} C_VEL
LIN {X 0,Y 594.322,Z 264.072,A -85,B 0,C 180,E1 -1248.955,E2 -1248.955} C_VEL
LIN {X 0,Y 594.341,Z 264.077,A -85,B 0,C 180,E1 -1251.841,E2 -1251.841} C_VEL
LIN {X 0,Y 594.331,Z 264.077,A -85,B 0,C 180,E1 -1253.89,E2 -1253.89} C_VEL
LIN {X 0,Y 594.319,Z 264.076,A -85,B 0,C 180,E1 -1255.93,E2 -1255.93} C_VEL
LIN {X 0,Y 594.358,Z 264.071,A -85,B 0,C 180,E1 -1257.966,E2 -1257.966} C_VEL
LIN {X 0,Y 594.374,Z 264.069,A -85,B 0,C 180,E1 -1259.999,E2 -1259.999} C_VEL
LIN {X 0,Y 594.355,Z 264.069,A -85,B 0,C 180,E1 -1262.71,E2 -1262.71} C_VEL
LIN {X 0,Y 594.365,Z 264.076,A -85,B 0,C 180,E1 -1265.427,E2 -1265.427} C_VEL
LIN {X 0,Y 594.328,Z 264.072,A -85,B 0,C 180,E1 -1268.157,E2 -1268.157} C_VEL
LIN {X 0,Y 594.352,Z 264.073,A -85,B 0,C 180,E1 -1271.06,E2 -1271.06} C_VEL
LIN {X 0,Y 594.316,Z 264.073,A -85,B 0,C 180,E1 -1274.149,E2 -1274.149} C_VEL
LIN {X 0,Y 594.316,Z 264.076,A -85,B 0,C 180,E1 -1275.271,E2 -1275.271} C_VEL
LIN {X 0,Y 593.641,Z 264.159,A -85,B 0,C 180,E1 -1275.837,E2 -1275.837} C_VEL
LIN {X 0,Y 590.775,Z 264.514,A -85,B 0,C 180,E1 -1276.754,E2 -1276.754} C_VEL
LIN {X 0,Y 588.365,Z 264.821,A -85,B 0,C 180,E1 -1277.493,E2 -1277.493} C_VEL
LIN {X 0,Y 587.342,Z 264.942,A -85,B 0,C 180,E1 -1278.063,E2 -1278.063} C_VEL
LIN {X 0,Y 587.264,Z 264.95,A -85,B 0,C 180,E1 -1278.256,E2 -1278.256} C_VEL
LIN {X 0,Y 587.318,Z 264.95,A -85,B 0,C 180,E1 -1281.036,E2 -1281.036} C_VEL
LIN {X 0,Y 587.269,Z 264.951,A -85,B 0,C 180,E1 -1284.008,E2 -1284.008} C_VEL
LIN {X 0,Y 587.285,Z 264.947,A -85,B 0,C 180,E1 -1286.279,E2 -1286.279} C_VEL
LIN {X 0,Y 587.323,Z 264.952,A -85,B 0,C 180,E1 -1289.13,E2 -1289.13} C_VEL
LIN {X 0,Y 587.327,Z 264.945,A -85,B 0,C 180,E1 -1291.834,E2 -1291.834} C_VEL
LIN {X 0,Y 587.315,Z 264.945,A -85,B 0,C 180,E1 -1294.344,E2 -1294.344} C_VEL
LIN {X 0,Y 587.323,Z 264.946,A -85,B 0,C 180,E1 -1297.607,E2 -1297.607} C_VEL
LIN {X 0,Y 587.292,Z 264.949,A -85,B 0,C 180,E1 -1300.254,E2 -1300.254} C_VEL
LIN {X 0,Y 587.287,Z 264.958,A -85,B 0,C 180,E1 -1303.116,E2 -1303.116} C_VEL
LIN {X 0,Y 587.279,Z 264.948,A -85,B 0,C 180,E1 -1306.046,E2 -1306.046} C_VEL
LIN {X 0,Y 587.316,Z 264.955,A -85,B 0,C 180,E1 -1308.924,E2 -1308.924} C_VEL
LIN {X 0,Y 587.302,Z 264.949,A -85,B 0,C 180,E1 -1311.519,E2 -1311.519} C_VEL
LIN {X 0,Y 587.273,Z 264.95,A -85,B 0,C 180,E1 -1314.099,E2 -1314.099} C_VEL
LIN {X 0,Y 587.308,Z 264.952,A -85,B 0,C 180,E1 -1316.602,E2 -1316.602} C_VEL
LIN {X 0,Y 587.315,Z 264.952,A -85,B 0,C 180,E1 -1319.033,E2 -1319.033} C_VEL
LIN {X 0,Y 587.3,Z 264.95,A -85,B 0,C 180,E1 -1321.402,E2 -1321.402} C_VEL
LIN {X 0,Y 587.316,Z 264.945,A -85,B 0,C 180,E1 -1323.823,E2 -1323.823} C_VEL
LIN {X 0,Y 587.301,Z 264.947,A -85,B 0,C 180,E1 -1325.992,E2 -1325.992} C_VEL
LIN {X 0,Y 587.296,Z 264.95,A -85,B 0,C 180,E1 -1328.225,E2 -1328.225} C_VEL
LIN {X 0,Y 587.33,Z 264.948,A -85,B 0,C 180,E1 -1331.151,E2 -1331.151} C_VEL
LIN {X 0,Y 587.301,Z 264.948,A -85,B 0,C 180,E1 -1334.024,E2 -1334.024} C_VEL
LIN {X 0,Y 587.332,Z 264.946,A -85,B 0,C 180,E1 -1336.154,E2 -1336.154} C_VEL
LIN {X 0,Y 587.394,Z 264.941,A -85,B 0,C 180,E1 -1338.963,E2 -1338.963} C_VEL
LIN {X 0,Y 587.361,Z 264.947,A -85,B 0,C 180,E1 -1342.437,E2 -1342.437} C_VEL
LIN {X 0,Y 587.343,Z 264.944,A -85,B 0,C 180,E1 -1345.195,E2 -1345.195} C_VEL
LIN {X 0,Y 587.335,Z 264.945,A -85,B 0,C 180,E1 -1347.943,E2 -1347.943} C_VEL
LIN {X 0,Y 587.388,Z 264.946,A -85,B 0,C 180,E1 -1350.685,E2 -1350.685} C_VEL
LIN {X 0,Y 587.311,Z 264.948,A -85,B 0,C 180,E1 -1353.43,E2 -1353.43} C_VEL
LIN {X 0,Y 587.336,Z 264.945,A -85,B 0,C 180,E1 -1355.493,E2 -1355.493} C_VEL
LIN {X 0,Y 587.368,Z 265.149,A -85,B 0,C 180,E1 -1357.131,E2 -1357.131} C_VEL
LIN {X 0,Y 587.85,Z 269.36,A -85,B 0,C 180,E1 -1357.729,E2 -1357.729} C_VEL
LIN {X 0,Y 587.734,Z 287.252,A -85,B 0,C 180,E1 -1360.158,E2 -1360.158} C_VEL
LIN {X 0,Y 587.725,Z 292.918,A -85,B 0,C 180,E1 -1360.921,E2 -1360.921} C_VEL
LIN {X 0,Y 588.548,Z 297.861,A -85,B 0,C 180,E1 -1361.014,E2 -1361.014} C_VEL
LIN {X 0,Y 588.29,Z 457.534,A -85,B 0,C 180,E1 -1363.031,E2 -1363.031} C_VEL
LIN {X 0,Y 588.225,Z 472.924,A -85,B 0,C 180,E1 -1363.362,E2 -1363.362} C_VEL
LIN {X 0,Y 588.098,Z 487.88,A -85,B 0,C 180,E1 -1363.827,E2 -1363.827} C_VEL
LIN {X 0,Y 587.959,Z 502.834,A -85,B 0,C 180,E1 -1364.448,E2 -1364.448} C_VEL
LIN {X 0,Y 587.826,Z 516.425,A -85,B 0,C 180,E1 -1365.161,E2 -1365.161} C_VEL
LIN {X 0,Y 587.677,Z 530.272,A -85,B 0,C 180,E1 -1366.054,E2 -1366.054} C_VEL
LIN {X 0,Y 587.586,Z 542.297,A -85,B 0,C 180,E1 -1366.994,E2 -1366.994} C_VEL
LIN {X 0,Y 587.444,Z 554.372,A -85,B 0,C 180,E1 -1368.122,E2 -1368.122} C_VEL
LIN {X 0,Y 587.352,Z 564.358,A -85,B 0,C 180,E1 -1369.24,E2 -1369.24} C_VEL
LIN {X 0,Y 587.311,Z 573.678,A -85,B 0,C 180,E1 -1370.485,E2 -1370.485} C_VEL
LIN {X 0,Y 587.232,Z 581.685,A -85,B 0,C 180,E1 -1371.777,E2 -1371.777} C_VEL
LIN {X 0,Y 587.205,Z 587.197,A -85,B 0,C 180,E1 -1372.847,E2 -1372.847} C_VEL
LIN {X 0,Y 587.212,Z 592.216,A -85,B 0,C 180,E1 -1374.011,E2 -1374.011} C_VEL
LIN {X 0,Y 587.145,Z 597.249,A -85,B 0,C 180,E1 -1375.525,E2 -1375.525} C_VEL
LIN {X 0,Y 587.116,Z 600.789,A -85,B 0,C 180,E1 -1377.056,E2 -1377.056} C_VEL
LIN {X 0,Y 587.131,Z 602.866,A -85,B 0,C 180,E1 -1378.606,E2 -1378.606} C_VEL
LIN {X 0,Y 587.142,Z 603.476,A -85,B 0,C 180,E1 -1380.18,E2 -1380.18} C_VEL
LIN {X 0,Y 587.136,Z 603.212,A -85,B 0,C 180,E1 -1380.977,E2 -1380.977} C_VEL
LIN {X 0,Y 587.117,Z 602.533,A -85,B 0,C 180,E1 -1381.804,E2 -1381.804} C_VEL
LIN {X 0,Y 587.127,Z 600.701,A -85,B 0,C 180,E1 -1383.084,E2 -1383.084} C_VEL
LIN {X 0,Y 587.162,Z 596.942,A -85,B 0,C 180,E1 -1384.669,E2 -1384.669} C_VEL
LIN {X 0,Y 587.207,Z 592.853,A -85,B 0,C 180,E1 -1385.905,E2 -1385.905} C_VEL
LIN {X 0,Y 587.191,Z 587.461,A -85,B 0,C 180,E1 -1387.186,E2 -1387.186} C_VEL
LIN {X 0,Y 587.245,Z 580.697,A -85,B 0,C 180,E1 -1388.485,E2 -1388.485} C_VEL
LIN {X 0,Y 587.286,Z 573.069,A -85,B 0,C 180,E1 -1389.693,E2 -1389.693} C_VEL
LIN {X 0,Y 587.376,Z 564.017,A -85,B 0,C 180,E1 -1390.89,E2 -1390.89} C_VEL
LIN {X 0,Y 587.46,Z 553.439,A -85,B 0,C 180,E1 -1392.062,E2 -1392.062} C_VEL
LIN {X 0,Y 587.58,Z 541.678,A -85,B 0,C 180,E1 -1393.149,E2 -1393.149} C_VEL
LIN {X 0,Y 587.722,Z 528.549,A -85,B 0,C 180,E1 -1394.156,E2 -1394.156} C_VEL
LIN {X 0,Y 587.838,Z 515.85,A -85,B 0,C 180,E1 -1394.963,E2 -1394.963} C_VEL
LIN {X 0,Y 587.988,Z 502.051,A -85,B 0,C 180,E1 -1395.679,E2 -1395.679} C_VEL
LIN {X 0,Y 588.131,Z 487.717,A -85,B 0,C 180,E1 -1396.267,E2 -1396.267} C_VEL
LIN {X 0,Y 588.216,Z 472.299,A -85,B 0,C 180,E1 -1396.745,E2 -1396.745} C_VEL
LIN {X 0,Y 588.309,Z 456.869,A -85,B 0,C 180,E1 -1397.07,E2 -1397.07} C_VEL
LIN {X 0,Y 588.458,Z 296.677,A -85,B 0,C 180,E1 -1399.094,E2 -1399.094} C_VEL
LIN {X 0,Y 587.709,Z 292.773,A -85,B 0,C 180,E1 -1399.189,E2 -1399.189} C_VEL
LIN {X 0,Y 587.869,Z 272.929,A -85,B 0,C 180,E1 -1401.871,E2 -1401.871} C_VEL
LIN {X 0,Y 587.783,Z 267.323,A -85,B 0,C 180,E1 -1402.643,E2 -1402.643} C_VEL
LIN {X 0,Y 587.36,Z 264.948,A -85,B 0,C 180,E1 -1402.988,E2 -1402.988} C_VEL
LIN {X 0,Y 587.355,Z 264.948,A -85,B 0,C 180,E1 -1405.782,E2 -1405.782} C_VEL
LIN {X 0,Y 587.341,Z 264.944,A -85,B 0,C 180,E1 -1408.233,E2 -1408.233} C_VEL
LIN {X 0,Y 587.339,Z 264.945,A -85,B 0,C 180,E1 -1410.866,E2 -1410.866} C_VEL
LIN {X 0,Y 587.345,Z 264.946,A -85,B 0,C 180,E1 -1413.819,E2 -1413.819} C_VEL
LIN {X 0,Y 587.309,Z 264.949,A -85,B 0,C 180,E1 -1416.742,E2 -1416.742} C_VEL
LIN {X 0,Y 587.32,Z 264.949,A -85,B 0,C 180,E1 -1419.696,E2 -1419.696} C_VEL
LIN {X 0,Y 587.346,Z 264.944,A -85,B 0,C 180,E1 -1422.595,E2 -1422.595} C_VEL
LIN {X 0,Y 587.349,Z 264.944,A -85,B 0,C 180,E1 -1425.74,E2 -1425.74} C_VEL
LIN {X 0,Y 587.332,Z 264.95,A -85,B 0,C 180,E1 -1428.867,E2 -1428.867} C_VEL
LIN {X 0,Y 587.325,Z 264.946,A -85,B 0,C 180,E1 -1431.745,E2 -1431.745} C_VEL
LIN {X 0,Y 587.351,Z 264.943,A -85,B 0,C 180,E1 -1434.508,E2 -1434.508} C_VEL
LIN {X 0,Y 587.355,Z 264.946,A -85,B 0,C 180,E1 -1437.258,E2 -1437.258} C_VEL
LIN {X 0,Y 587.355,Z 264.941,A -85,B 0,C 180,E1 -1440.001,E2 -1440.001} C_VEL
LIN {X 0,Y 587.372,Z 264.946,A -85,B 0,C 180,E1 -1442.744,E2 -1442.744} C_VEL
LIN {X 0,Y 587.327,Z 264.945,A -85,B 0,C 180,E1 -1445.494,E2 -1445.494} C_VEL
LIN {X 0,Y 587.326,Z 264.944,A -85,B 0,C 180,E1 -1447.565,E2 -1447.565} C_VEL
LIN {X 0,Y 587.325,Z 264.948,A -85,B 0,C 180,E1 -1450.341,E2 -1450.341} C_VEL
LIN {X 0,Y 587.294,Z 264.951,A -85,B 0,C 180,E1 -1453.143,E2 -1453.143} C_VEL
LIN {X 0,Y 587.308,Z 264.948,A -85,B 0,C 180,E1 -1455.265,E2 -1455.265} C_VEL
LIN {X 0,Y 587.328,Z 264.944,A -85,B 0,C 180,E1 -1457.407,E2 -1457.407} C_VEL
LIN {X 0,Y 587.292,Z 264.948,A -85,B 0,C 180,E1 -1459.578,E2 -1459.578} C_VEL
LIN {X 0,Y 587.298,Z 264.949,A -85,B 0,C 180,E1 -1461.776,E2 -1461.776} C_VEL
LIN {X 0,Y 587.295,Z 264.954,A -85,B 0,C 180,E1 -1464.762,E2 -1464.762} C_VEL
LIN {X 0,Y 587.29,Z 264.95,A -85,B 0,C 180,E1 -1467.684,E2 -1467.684} C_VEL
LIN {X 0,Y 587.299,Z 264.954,A -85,B 0,C 180,E1 -1470.173,E2 -1470.173} C_VEL
LIN {X 0,Y 587.318,Z 264.946,A -85,B 0,C 180,E1 -1473.111,E2 -1473.111} C_VEL
LIN {X 0,Y 587.262,Z 264.957,A -85,B 0,C 180,E1 -1475.903,E2 -1475.903} C_VEL
LIN {X 0,Y 587.301,Z 264.953,A -85,B 0,C 180,E1 -1478.482,E2 -1478.482} C_VEL
LIN {X 0,Y 587.28,Z 264.95,A -85,B 0,C 180,E1 -1481.162,E2 -1481.162} C_VEL
LIN {X 0,Y 587.296,Z 264.958,A -85,B 0,C 180,E1 -1484.112,E2 -1484.112} C_VEL
LIN {X 0,Y 587.271,Z 264.952,A -85,B 0,C 180,E1 -1486.991,E2 -1486.991} C_VEL
LIN {X 0,Y 587.296,Z 264.954,A -85,B 0,C 180,E1 -1489.746,E2 -1489.746} C_VEL
LIN {X 0,Y 587.312,Z 264.949,A -85,B 0,C 180,E1 -1492.391,E2 -1492.391} C_VEL
LIN {X 0,Y 587.331,Z 264.95,A -85,B 0,C 180,E1 -1495.655,E2 -1495.655} C_VEL
LIN {X 0,Y 587.328,Z 264.949,A -85,B 0,C 180,E1 -1498.231,E2 -1498.231} C_VEL
LIN {X 0,Y 587.34,Z 264.944,A -85,B 0,C 180,E1 -1500.869,E2 -1500.869} C_VEL
LIN {X 0,Y 587.323,Z 264.978,A -85,B 0,C 180,E1 -1504.078,E2 -1504.078} C_VEL
LIN {X 0,Y 588.241,Z 270.024,A -85,B 0,C 180,E1 -1504.735,E2 -1504.735} C_VEL
LIN {X 0,Y 588.053,Z 293.277,A -85,B 0,C 180,E1 -1507.516,E2 -1507.516} C_VEL
LIN {X 0,Y 587.845,Z 318.247,A -85,B 0,C 180,E1 -1510.443,E2 -1510.443} C_VEL
LIN {X 0,Y 587.814,Z 322.083,A -85,B 0,C 180,E1 -1510.871,E2 -1510.871} C_VEL
LIN {X 0,Y 588.594,Z 326.614,A -85,B 0,C 180,E1 -1510.955,E2 -1510.955} C_VEL
LIN {X 0,Y 588.305,Z 488.302,A -85,B 0,C 180,E1 -1512.998,E2 -1512.998} C_VEL
LIN {X 0,Y 588.222,Z 503.732,A -85,B 0,C 180,E1 -1513.337,E2 -1513.337} C_VEL
LIN {X 0,Y 588.071,Z 519.061,A -85,B 0,C 180,E1 -1513.824,E2 -1513.824} C_VEL
LIN {X 0,Y 587.988,Z 532.78,A -85,B 0,C 180,E1 -1514.4,E2 -1514.4} C_VEL
LIN {X 0,Y 587.836,Z 546.25,A -85,B 0,C 180,E1 -1515.106,E2 -1515.106} C_VEL
LIN {X 0,Y 587.74,Z 559.123,A -85,B 0,C 180,E1 -1515.93,E2 -1515.93} C_VEL
LIN {X 0,Y 587.583,Z 571.294,A -85,B 0,C 180,E1 -1516.865,E2 -1516.865} C_VEL
LIN {X 0,Y 587.453,Z 582.754,A -85,B 0,C 180,E1 -1517.916,E2 -1517.916} C_VEL
LIN {X 0,Y 587.349,Z 592.394,A -85,B 0,C 180,E1 -1518.963,E2 -1518.963} C_VEL
LIN {X 0,Y 587.304,Z 601.86,A -85,B 0,C 180,E1 -1520.182,E2 -1520.182} C_VEL
LIN {X 0,Y 587.264,Z 609.734,A -85,B 0,C 180,E1 -1521.397,E2 -1521.397} C_VEL
LIN {X 0,Y 587.215,Z 617.091,A -85,B 0,C 180,E1 -1522.781,E2 -1522.781} C_VEL
LIN {X 0,Y 587.224,Z 622.925,A -85,B 0,C 180,E1 -1524.162,E2 -1524.162} C_VEL
LIN {X 0,Y 587.136,Z 626.385,A -85,B 0,C 180,E1 -1525.194,E2 -1525.194} C_VEL
LIN {X 0,Y 587.179,Z 629.888,A -85,B 0,C 180,E1 -1526.569,E2 -1526.569} C_VEL
LIN {X 0,Y 587.138,Z 632.194,A -85,B 0,C 180,E1 -1527.942,E2 -1527.942} C_VEL
LIN {X 0,Y 587.137,Z 633.35,A -85,B 0,C 180,E1 -1529.314,E2 -1529.314} C_VEL
LIN {X 0,Y 587.137,Z 633.349,A -85,B 0,C 180,E1 -1530.686,E2 -1530.686} C_VEL
LIN {X 0,Y 587.138,Z 632.192,A -85,B 0,C 180,E1 -1532.058,E2 -1532.058} C_VEL
LIN {X 0,Y 587.179,Z 629.886,A -85,B 0,C 180,E1 -1533.431,E2 -1533.431} C_VEL
LIN {X 0,Y 587.136,Z 626.384,A -85,B 0,C 180,E1 -1534.807,E2 -1534.807} C_VEL
LIN {X 0,Y 587.178,Z 621.607,A -85,B 0,C 180,E1 -1536.184,E2 -1536.184} C_VEL
LIN {X 0,Y 587.23,Z 615.423,A -85,B 0,C 180,E1 -1537.565,E2 -1537.565} C_VEL
LIN {X 0,Y 587.267,Z 607.65,A -85,B 0,C 180,E1 -1538.95,E2 -1538.95} C_VEL
LIN {X 0,Y 587.351,Z 599.369,A -85,B 0,C 180,E1 -1540.166,E2 -1540.166} C_VEL
LIN {X 0,Y 587.4,Z 589.394,A -85,B 0,C 180,E1 -1541.386,E2 -1541.386} C_VEL
LIN {X 0,Y 587.522,Z 579.19,A -85,B 0,C 180,E1 -1542.434,E2 -1542.434} C_VEL
LIN {X 0,Y 587.629,Z 567.018,A -85,B 0,C 180,E1 -1543.487,E2 -1543.487} C_VEL
LIN {X 0,Y 587.775,Z 554.058,A -85,B 0,C 180,E1 -1544.416,E2 -1544.416} C_VEL
LIN {X 0,Y 587.888,Z 539.867,A -85,B 0,C 180,E1 -1545.248,E2 -1545.248} C_VEL
LIN {X 0,Y 588.051,Z 525.798,A -85,B 0,C 180,E1 -1545.91,E2 -1545.91} C_VEL
LIN {X 0,Y 588.171,Z 511.305,A -85,B 0,C 180,E1 -1546.442,E2 -1546.442} C_VEL
LIN {X 0,Y 588.281,Z 496.27,A -85,B 0,C 180,E1 -1546.845,E2 -1546.845} C_VEL
LIN {X 0,Y 588.323,Z 481.068,A -85,B 0,C 180,E1 -1547.11,E2 -1547.11} C_VEL
LIN {X 0,Y 588.503,Z 325.516,A -85,B 0,C 180,E1 -1549.062,E2 -1549.062} C_VEL
LIN {X 0,Y 587.797,Z 321.798,A -85,B 0,C 180,E1 -1549.145,E2 -1549.145} C_VEL
LIN {X 0,Y 588.033,Z 296.393,A -85,B 0,C 180,E1 -1552.116,E2 -1552.116} C_VEL
LIN {X 0,Y 588.234,Z 273.141,A -85,B 0,C 180,E1 -1554.888,E2 -1554.888} C_VEL
LIN {X 0,Y 588.08,Z 268.302,A -85,B 0,C 180,E1 -1555.482,E2 -1555.482} C_VEL
LIN {X 0,Y 587.33,Z 264.953,A -85,B 0,C 180,E1 -1555.948,E2 -1555.948} C_VEL
LIN {X 0,Y 587.343,Z 264.944,A -85,B 0,C 180,E1 -1559.132,E2 -1559.132} C_VEL
LIN {X 0,Y 587.339,Z 264.948,A -85,B 0,C 180,E1 -1561.834,E2 -1561.834} C_VEL
LIN {X 0,Y 587.329,Z 264.952,A -85,B 0,C 180,E1 -1564.345,E2 -1564.345} C_VEL
LIN {X 0,Y 587.318,Z 264.949,A -85,B 0,C 180,E1 -1567.609,E2 -1567.609} C_VEL
LIN {X 0,Y 587.302,Z 264.955,A -85,B 0,C 180,E1 -1570.255,E2 -1570.255} C_VEL
LIN {X 0,Y 587.283,Z 264.949,A -85,B 0,C 180,E1 -1573.114,E2 -1573.114} C_VEL
LIN {X 0,Y 587.297,Z 264.958,A -85,B 0,C 180,E1 -1576.046,E2 -1576.046} C_VEL
LIN {X 0,Y 587.303,Z 264.948,A -85,B 0,C 180,E1 -1578.84,E2 -1578.84} C_VEL
LIN {X 0,Y 587.31,Z 264.949,A -85,B 0,C 180,E1 -1581.518,E2 -1581.518} C_VEL
LIN {X 0,Y 587.272,Z 264.958,A -85,B 0,C 180,E1 -1584.098,E2 -1584.098} C_VEL
LIN {X 0,Y 587.33,Z 264.943,A -85,B 0,C 180,E1 -1586.888,E2 -1586.888} C_VEL
LIN {X 0,Y 587.317,Z 264.949,A -85,B 0,C 180,E1 -1589.492,E2 -1589.492} C_VEL
LIN {X 0,Y 587.297,Z 264.952,A -85,B 0,C 180,E1 -1592.179,E2 -1592.179} C_VEL
LIN {X 0,Y 587.287,Z 264.951,A -85,B 0,C 180,E1 -1594.48,E2 -1594.48} C_VEL
LIN {X 0,Y 587.301,Z 264.949,A -85,B 0,C 180,E1 -1597.133,E2 -1597.133} C_VEL
LIN {X 0,Y 587.311,Z 264.956,A -85,B 0,C 180,E1 -1599.694,E2 -1599.694} C_VEL
LIN {X 0,Y 587.274,Z 264.959,A -85,B 0,C 180,E1 -1601.871,E2 -1601.871} C_VEL
LIN {X 0,Y 587.293,Z 264.953,A -85,B 0,C 180,E1 -1604.023,E2 -1604.023} C_VEL
LIN {X 0,Y 587.326,Z 264.945,A -85,B 0,C 180,E1 -1606.153,E2 -1606.153} C_VEL
LIN {X 0,Y 587.282,Z 264.949,A -85,B 0,C 180,E1 -1608.96,E2 -1608.96} C_VEL
LIN {X 0,Y 587.308,Z 264.955,A -85,B 0,C 180,E1 -1611.743,E2 -1611.743} C_VEL
LIN {X 0,Y 587.291,Z 264.955,A -85,B 0,C 180,E1 -1613.816,E2 -1613.816} C_VEL
LIN {X 0,Y 587.275,Z 264.953,A -85,B 0,C 180,E1 -1615.881,E2 -1615.881} C_VEL
LIN {X 0,Y 587.332,Z 264.946,A -85,B 0,C 180,E1 -1617.942,E2 -1617.942} C_VEL
LIN {X 0,Y 587.345,Z 264.945,A -85,B 0,C 180,E1 -1619.999,E2 -1619.999} C_VEL
LIN {X 0,Y 587.326,Z 264.945,A -85,B 0,C 180,E1 -1622.742,E2 -1622.742} C_VEL
LIN {X 0,Y 587.328,Z 264.951,A -85,B 0,C 180,E1 -1625.492,E2 -1625.492} C_VEL
LIN {X 0,Y 587.292,Z 264.947,A -85,B 0,C 180,E1 -1628.255,E2 -1628.255} C_VEL
LIN {X 0,Y 587.319,Z 264.95,A -85,B 0,C 180,E1 -1631.123,E2 -1631.123} C_VEL
LIN {X 0,Y 587.287,Z 264.948,A -85,B 0,C 180,E1 -1634.234,E2 -1634.234} C_VEL
LIN {X 0,Y 587.303,Z 264.946,A -85,B 0,C 180,E1 -1636.802,E2 -1636.802} C_VEL
LIN {X 0,Y 587.264,Z 264.95,A -85,B 0,C 180,E1 -1638.256,E2 -1638.256} C_VEL
LIN {X 0,Y 586.629,Z 265.033,A -85,B 0,C 180,E1 -1638.828,E2 -1638.828} C_VEL
LIN {X 0,Y 583.832,Z 265.383,A -85,B 0,C 180,E1 -1639.757,E2 -1639.757} C_VEL
LIN {X 0,Y 581.435,Z 265.68,A -85,B 0,C 180,E1 -1640.504,E2 -1640.504} C_VEL
LIN {X 0,Y 580.374,Z 265.816,A -85,B 0,C 180,E1 -1641.08,E2 -1641.08} C_VEL
LIN {X 0,Y 580.272,Z 265.832,A -85,B 0,C 180,E1 -1641.276,E2 -1641.276} C_VEL
LIN {X 0,Y 580.234,Z 265.833,A -85,B 0,C 180,E1 -1643.558,E2 -1643.558} C_VEL
LIN {X 0,Y 580.245,Z 265.823,A -85,B 0,C 180,E1 -1646.327,E2 -1646.327} C_VEL
LIN {X 0,Y 580.253,Z 265.834,A -85,B 0,C 180,E1 -1649.303,E2 -1649.303} C_VEL
LIN {X 0,Y 580.278,Z 265.822,A -85,B 0,C 180,E1 -1652.2,E2 -1652.2} C_VEL
LIN {X 0,Y 580.261,Z 265.827,A -85,B 0,C 180,E1 -1654.696,E2 -1654.696} C_VEL
LIN {X 0,Y 580.27,Z 265.83,A -85,B 0,C 180,E1 -1657.268,E2 -1657.268} C_VEL
LIN {X 0,Y 580.272,Z 265.823,A -85,B 0,C 180,E1 -1660.269,E2 -1660.269} C_VEL
LIN {X 0,Y 580.251,Z 265.829,A -85,B 0,C 180,E1 -1663.389,E2 -1663.389} C_VEL
LIN {X 0,Y 580.223,Z 265.828,A -85,B 0,C 180,E1 -1666.338,E2 -1666.338} C_VEL
LIN {X 0,Y 580.277,Z 265.83,A -85,B 0,C 180,E1 -1669.155,E2 -1669.155} C_VEL
LIN {X 0,Y 580.267,Z 265.823,A -85,B 0,C 180,E1 -1671.927,E2 -1671.927} C_VEL
LIN {X 0,Y 580.237,Z 265.829,A -85,B 0,C 180,E1 -1674.452,E2 -1674.452} C_VEL
LIN {X 0,Y 580.269,Z 265.833,A -85,B 0,C 180,E1 -1676.974,E2 -1676.974} C_VEL
LIN {X 0,Y 580.271,Z 265.824,A -85,B 0,C 180,E1 -1679.424,E2 -1679.424} C_VEL
LIN {X 0,Y 580.277,Z 265.823,A -85,B 0,C 180,E1 -1682.141,E2 -1682.141} C_VEL
LIN {X 0,Y 580.301,Z 265.822,A -85,B 0,C 180,E1 -1685.269,E2 -1685.269} C_VEL
LIN {X 0,Y 580.248,Z 265.827,A -85,B 0,C 180,E1 -1687.947,E2 -1687.947} C_VEL
LIN {X 0,Y 580.299,Z 265.828,A -85,B 0,C 180,E1 -1690.914,E2 -1690.914} C_VEL
LIN {X 0,Y 580.254,Z 265.825,A -85,B 0,C 180,E1 -1693.825,E2 -1693.825} C_VEL
LIN {X 0,Y 580.298,Z 265.821,A -85,B 0,C 180,E1 -1695.982,E2 -1695.982} C_VEL
LIN {X 0,Y 580.332,Z 265.823,A -85,B 0,C 180,E1 -1698.827,E2 -1698.827} C_VEL
LIN {X 0,Y 580.29,Z 265.821,A -85,B 0,C 180,E1 -1701.643,E2 -1701.643} C_VEL
LIN {X 0,Y 580.311,Z 265.826,A -85,B 0,C 180,E1 -1704.44,E2 -1704.44} C_VEL
LIN {X 0,Y 580.321,Z 265.819,A -85,B 0,C 180,E1 -1707.223,E2 -1707.223} C_VEL
LIN {X 0,Y 580.322,Z 265.82,A -85,B 0,C 180,E1 -1710,E2 -1710} C_VEL
LIN {X 0,Y 580.336,Z 265.823,A -85,B 0,C 180,E1 -1712.776,E2 -1712.776} C_VEL
LIN {X 0,Y 580.302,Z 265.822,A -85,B 0,C 180,E1 -1715.56,E2 -1715.56} C_VEL
LIN {X 0,Y 580.335,Z 265.997,A -85,B 0,C 180,E1 -1716.955,E2 -1716.955} C_VEL
LIN {X 0,Y 580.961,Z 270.774,A -85,B 0,C 180,E1 -1717.647,E2 -1717.647} C_VEL
LIN {X 0,Y 580.811,Z 288.668,A -85,B 0,C 180,E1 -1720.105,E2 -1720.105} C_VEL
LIN {X 0,Y 580.765,Z 292.886,A -85,B 0,C 180,E1 -1720.678,E2 -1720.678} C_VEL
LIN {X 0,Y 581.824,Z 298.252,A -85,B 0,C 180,E1 -1720.791,E2 -1720.791} C_VEL
LIN {X 0,Y 581.496,Z 457.772,A -85,B 0,C 180,E1 -1722.831,E2 -1722.831} C_VEL
LIN {X 0,Y 581.424,Z 473.069,A -85,B 0,C 180,E1 -1723.166,E2 -1723.166} C_VEL
LIN {X 0,Y 581.251,Z 488.029,A -85,B 0,C 180,E1 -1723.637,E2 -1723.637} C_VEL
LIN {X 0,Y 581.097,Z 502.731,A -85,B 0,C 180,E1 -1724.254,E2 -1724.254} C_VEL
LIN {X 0,Y 580.929,Z 516.524,A -85,B 0,C 180,E1 -1724.986,E2 -1724.986} C_VEL
LIN {X 0,Y 580.777,Z 529.077,A -85,B 0,C 180,E1 -1725.799,E2 -1725.799} C_VEL
LIN {X 0,Y 580.612,Z 541.862,A -85,B 0,C 180,E1 -1726.797,E2 -1726.797} C_VEL
LIN {X 0,Y 580.453,Z 552.65,A -85,B 0,C 180,E1 -1727.801,E2 -1727.801} C_VEL
LIN {X 0,Y 580.364,Z 562.635,A -85,B 0,C 180,E1 -1728.9,E2 -1728.9} C_VEL
LIN {X 0,Y 580.274,Z 572.468,A -85,B 0,C 180,E1 -1730.192,E2 -1730.192} C_VEL
LIN {X 0,Y 580.179,Z 580.658,A -85,B 0,C 180,E1 -1731.495,E2 -1731.495} C_VEL
LIN {X 0,Y 580.113,Z 588.183,A -85,B 0,C 180,E1 -1732.972,E2 -1732.972} C_VEL
LIN {X 0,Y 580.103,Z 593.604,A -85,B 0,C 180,E1 -1734.324,E2 -1734.324} C_VEL
LIN {X 0,Y 580.036,Z 598.25,A -85,B 0,C 180,E1 -1735.86,E2 -1735.86} C_VEL
LIN {X 0,Y 580.04,Z 601.415,A -85,B 0,C 180,E1 -1737.413,E2 -1737.413} C_VEL
LIN {X 0,Y 580.041,Z 603.136,A -85,B 0,C 180,E1 -1738.989,E2 -1738.989} C_VEL
LIN {X 0,Y 580.053,Z 603.384,A -85,B 0,C 180,E1 -1740.588,E2 -1740.588} C_VEL
LIN {X 0,Y 580.022,Z 602.092,A -85,B 0,C 180,E1 -1742.217,E2 -1742.217} C_VEL
LIN {X 0,Y 580.048,Z 600.374,A -85,B 0,C 180,E1 -1743.281,E2 -1743.281} C_VEL
LIN {X 0,Y 580.073,Z 596.989,A -85,B 0,C 180,E1 -1744.71,E2 -1744.71} C_VEL
LIN {X 0,Y 580.111,Z 592.594,A -85,B 0,C 180,E1 -1746.05,E2 -1746.05} C_VEL
LIN {X 0,Y 580.127,Z 587.434,A -85,B 0,C 180,E1 -1747.28,E2 -1747.28} C_VEL
LIN {X 0,Y 580.169,Z 580.65,A -85,B 0,C 180,E1 -1748.597,E2 -1748.597} C_VEL
LIN {X 0,Y 580.231,Z 572.203,A -85,B 0,C 180,E1 -1749.937,E2 -1749.937} C_VEL
LIN {X 0,Y 580.368,Z 562.428,A -85,B 0,C 180,E1 -1751.214,E2 -1751.214} C_VEL
LIN {X 0,Y 580.472,Z 551.589,A -85,B 0,C 180,E1 -1752.395,E2 -1752.395} C_VEL
LIN {X 0,Y 580.619,Z 539.497,A -85,B 0,C 180,E1 -1753.493,E2 -1753.493} C_VEL
LIN {X 0,Y 580.822,Z 526.807,A -85,B 0,C 180,E1 -1754.449,E2 -1754.449} C_VEL
LIN {X 0,Y 580.968,Z 513.294,A -85,B 0,C 180,E1 -1755.29,E2 -1755.29} C_VEL
LIN {X 0,Y 581.16,Z 498.85,A -85,B 0,C 180,E1 -1756.015,E2 -1756.015} C_VEL
LIN {X 0,Y 581.307,Z 484.906,A -85,B 0,C 180,E1 -1756.563,E2 -1756.563} C_VEL
LIN {X 0,Y 581.454,Z 470.149,A -85,B 0,C 180,E1 -1756.999,E2 -1756.999} C_VEL
LIN {X 0,Y 581.544,Z 454.694,A -85,B 0,C 180,E1 -1757.308,E2 -1757.308} C_VEL
LIN {X 0,Y 581.785,Z 297.967,A -85,B 0,C 180,E1 -1759.304,E2 -1759.304} C_VEL
LIN {X 0,Y 580.759,Z 292.78,A -85,B 0,C 180,E1 -1759.426,E2 -1759.426} C_VEL
LIN {X 0,Y 580.959,Z 273.051,A -85,B 0,C 180,E1 -1762.128,E2 -1762.128} C_VEL
LIN {X 0,Y 580.83,Z 268.438,A -85,B 0,C 180,E1 -1762.774,E2 -1762.774} C_VEL
LIN {X 0,Y 580.316,Z 265.826,A -85,B 0,C 180,E1 -1763.17,E2 -1763.17} C_VEL
LIN {X 0,Y 580.306,Z 265.822,A -85,B 0,C 180,E1 -1766.147,E2 -1766.147} C_VEL
LIN {X 0,Y 580.276,Z 265.824,A -85,B 0,C 180,E1 -1768.617,E2 -1768.617} C_VEL
LIN {X 0,Y 580.283,Z 265.826,A -85,B 0,C 180,E1 -1771.025,E2 -1771.025} C_VEL
LIN {X 0,Y 580.312,Z 265.825,A -85,B 0,C 180,E1 -1773.659,E2 -1773.659} C_VEL
LIN {X 0,Y 580.265,Z 265.825,A -85,B 0,C 180,E1 -1776.443,E2 -1776.443} C_VEL
LIN {X 0,Y 580.269,Z 265.832,A -85,B 0,C 180,E1 -1779.439,E2 -1779.439} C_VEL
LIN {X 0,Y 580.268,Z 265.828,A -85,B 0,C 180,E1 -1781.647,E2 -1781.647} C_VEL
LIN {X 0,Y 580.265,Z 265.826,A -85,B 0,C 180,E1 -1783.827,E2 -1783.827} C_VEL
LIN {X 0,Y 580.312,Z 265.819,A -85,B 0,C 180,E1 -1785.984,E2 -1785.984} C_VEL
LIN {X 0,Y 580.289,Z 265.826,A -85,B 0,C 180,E1 -1788.828,E2 -1788.828} C_VEL
LIN {X 0,Y 580.295,Z 265.822,A -85,B 0,C 180,E1 -1791.645,E2 -1791.645} C_VEL
LIN {X 0,Y 580.314,Z 265.819,A -85,B 0,C 180,E1 -1794.441,E2 -1794.441} C_VEL
LIN {X 0,Y 580.323,Z 265.823,A -85,B 0,C 180,E1 -1797.225,E2 -1797.225} C_VEL
LIN {X 0,Y 580.326,Z 265.816,A -85,B 0,C 180,E1 -1800.001,E2 -1800.001} C_VEL
LIN {X 0,Y 580.336,Z 265.823,A -85,B 0,C 180,E1 -1802.778,E2 -1802.778} C_VEL
LIN {X 0,Y 580.294,Z 265.821,A -85,B 0,C 180,E1 -1805.561,E2 -1805.561} C_VEL
LIN {X 0,Y 580.275,Z 265.822,A -85,B 0,C 180,E1 -1807.657,E2 -1807.657} C_VEL
LIN {X 0,Y 580.287,Z 265.827,A -85,B 0,C 180,E1 -1810.468,E2 -1810.468} C_VEL
LIN {X 0,Y 580.249,Z 265.827,A -85,B 0,C 180,E1 -1813.306,E2 -1813.306} C_VEL
LIN {X 0,Y 580.274,Z 265.823,A -85,B 0,C 180,E1 -1815.454,E2 -1815.454} C_VEL
LIN {X 0,Y 580.273,Z 265.823,A -85,B 0,C 180,E1 -1817.626,E2 -1817.626} C_VEL
LIN {X 0,Y 580.27,Z 265.824,A -85,B 0,C 180,E1 -1819.824,E2 -1819.824} C_VEL
LIN {X 0,Y 580.251,Z 265.829,A -85,B 0,C 180,E1 -1822.054,E2 -1822.054} C_VEL
LIN {X 0,Y 580.254,Z 265.831,A -85,B 0,C 180,E1 -1824.719,E2 -1824.719} C_VEL
LIN {X 0,Y 580.234,Z 265.828,A -85,B 0,C 180,E1 -1827.405,E2 -1827.405} C_VEL
LIN {X 0,Y 580.251,Z 265.827,A -85,B 0,C 180,E1 -1829.775,E2 -1829.775} C_VEL
LIN {X 0,Y 580.276,Z 265.83,A -85,B 0,C 180,E1 -1832.203,E2 -1832.203} C_VEL
LIN {X 0,Y 580.259,Z 265.829,A -85,B 0,C 180,E1 -1834.699,E2 -1834.699} C_VEL
LIN {X 0,Y 580.256,Z 265.825,A -85,B 0,C 180,E1 -1837.272,E2 -1837.272} C_VEL
LIN {X 0,Y 580.261,Z 265.834,A -85,B 0,C 180,E1 -1840.269,E2 -1840.269} C_VEL
LIN {X 0,Y 580.248,Z 265.828,A -85,B 0,C 180,E1 -1842.71,E2 -1842.71} C_VEL
LIN {X 0,Y 580.244,Z 265.83,A -85,B 0,C 180,E1 -1845.612,E2 -1845.612} C_VEL
LIN {X 0,Y 580.237,Z 265.835,A -85,B 0,C 180,E1 -1848.229,E2 -1848.229} C_VEL
LIN {X 0,Y 580.259,Z 265.825,A -85,B 0,C 180,E1 -1850.965,E2 -1850.965} C_VEL
LIN {X 0,Y 580.234,Z 265.832,A -85,B 0,C 180,E1 -1853.595,E2 -1853.595} C_VEL
LIN {X 0,Y 580.304,Z 265.826,A -85,B 0,C 180,E1 -1856.146,E2 -1856.146} C_VEL
LIN {X 0,Y 580.265,Z 265.826,A -85,B 0,C 180,E1 -1858.615,E2 -1858.615} C_VEL
LIN {X 0,Y 580.282,Z 265.824,A -85,B 0,C 180,E1 -1861.024,E2 -1861.024} C_VEL
LIN {X 0,Y 580.282,Z 265.855,A -85,B 0,C 180,E1 -1863.856,E2 -1863.856} C_VEL
LIN {X 0,Y 581.411,Z 271.428,A -85,B 0,C 180,E1 -1864.589,E2 -1864.589} C_VEL
LIN {X 0,Y 581.244,Z 291.891,A -85,B 0,C 180,E1 -1867.071,E2 -1867.071} C_VEL
LIN {X 0,Y 580.967,Z 316.686,A -85,B 0,C 180,E1 -1870.018,E2 -1870.018} C_VEL
LIN {X 0,Y 580.896,Z 321.911,A -85,B 0,C 180,E1 -1870.631,E2 -1870.631} C_VEL
LIN {X 0,Y 581.879,Z 327.796,A -85,B 0,C 180,E1 -1870.742,E2 -1870.742} C_VEL
LIN {X 0,Y 581.53,Z 487.827,A -85,B 0,C 180,E1 -1872.786,E2 -1872.786} C_VEL
LIN {X 0,Y 581.423,Z 503.078,A -85,B 0,C 180,E1 -1873.119,E2 -1873.119} C_VEL
LIN {X 0,Y 581.259,Z 517.814,A -85,B 0,C 180,E1 -1873.584,E2 -1873.584} C_VEL
LIN {X 0,Y 581.124,Z 532.782,A -85,B 0,C 180,E1 -1874.211,E2 -1874.211} C_VEL
LIN {X 0,Y 580.944,Z 546.253,A -85,B 0,C 180,E1 -1874.925,E2 -1874.925} C_VEL
LIN {X 0,Y 580.804,Z 559.489,A -85,B 0,C 180,E1 -1875.784,E2 -1875.784} C_VEL
LIN {X 0,Y 580.608,Z 571.296,A -85,B 0,C 180,E1 -1876.704,E2 -1876.704} C_VEL
LIN {X 0,Y 580.479,Z 582.754,A -85,B 0,C 180,E1 -1877.768,E2 -1877.768} C_VEL
LIN {X 0,Y 580.308,Z 593.457,A -85,B 0,C 180,E1 -1878.954,E2 -1878.954} C_VEL
LIN {X 0,Y 580.268,Z 601.861,A -85,B 0,C 180,E1 -1880.062,E2 -1880.062} C_VEL
LIN {X 0,Y 580.214,Z 609.735,A -85,B 0,C 180,E1 -1881.292,E2 -1881.292} C_VEL
LIN {X 0,Y 580.131,Z 617.091,A -85,B 0,C 180,E1 -1882.692,E2 -1882.692} C_VEL
LIN {X 0,Y 580.129,Z 622.925,A -85,B 0,C 180,E1 -1884.09,E2 -1884.09} C_VEL
LIN {X 0,Y 580.041,Z 626.386,A -85,B 0,C 180,E1 -1885.135,E2 -1885.135} C_VEL
LIN {X 0,Y 580.104,Z 629.889,A -85,B 0,C 180,E1 -1886.528,E2 -1886.528} C_VEL
LIN {X 0,Y 580.037,Z 632.193,A -85,B 0,C 180,E1 -1887.917,E2 -1887.917} C_VEL
LIN {X 0,Y 580.038,Z 633.349,A -85,B 0,C 180,E1 -1889.306,E2 -1889.306} C_VEL
LIN {X 0,Y 580.038,Z 633.349,A -85,B 0,C 180,E1 -1890.695,E2 -1890.695} C_VEL
LIN {X 0,Y 580.037,Z 632.191,A -85,B 0,C 180,E1 -1892.083,E2 -1892.083} C_VEL
LIN {X 0,Y 580.105,Z 629.886,A -85,B 0,C 180,E1 -1893.473,E2 -1893.473} C_VEL
LIN {X 0,Y 580.041,Z 626.384,A -85,B 0,C 180,E1 -1894.866,E2 -1894.866} C_VEL
LIN {X 0,Y 580.091,Z 621.608,A -85,B 0,C 180,E1 -1896.26,E2 -1896.26} C_VEL
LIN {X 0,Y 580.166,Z 615.423,A -85,B 0,C 180,E1 -1897.658,E2 -1897.658} C_VEL
LIN {X 0,Y 580.208,Z 607.649,A -85,B 0,C 180,E1 -1899.06,E2 -1899.06} C_VEL
LIN {X 0,Y 580.309,Z 599.369,A -85,B 0,C 180,E1 -1900.29,E2 -1900.29} C_VEL
LIN {X 0,Y 580.383,Z 589.394,A -85,B 0,C 180,E1 -1901.525,E2 -1901.525} C_VEL
LIN {X 0,Y 580.541,Z 579.189,A -85,B 0,C 180,E1 -1902.586,E2 -1902.586} C_VEL
LIN {X 0,Y 580.678,Z 567.019,A -85,B 0,C 180,E1 -1903.651,E2 -1903.651} C_VEL
LIN {X 0,Y 580.875,Z 553.528,A -85,B 0,C 180,E1 -1904.625,E2 -1904.625} C_VEL
LIN {X 0,Y 581.019,Z 539.87,A -85,B 0,C 180,E1 -1905.433,E2 -1905.433} C_VEL
LIN {X 0,Y 581.206,Z 525.799,A -85,B 0,C 180,E1 -1906.103,E2 -1906.103} C_VEL
LIN {X 0,Y 581.359,Z 511.306,A -85,B 0,C 180,E1 -1906.64,E2 -1906.64} C_VEL
LIN {X 0,Y 581.489,Z 496.05,A -85,B 0,C 180,E1 -1907.052,E2 -1907.052} C_VEL
LIN {X 0,Y 581.553,Z 480.528,A -85,B 0,C 180,E1 -1907.323,E2 -1907.323} C_VEL
LIN {X 0,Y 581.809,Z 326.568,A -85,B 0,C 180,E1 -1909.277,E2 -1909.277} C_VEL
LIN {X 0,Y 580.896,Z 321.777,A -85,B 0,C 180,E1 -1909.384,E2 -1909.384} C_VEL
LIN {X 0,Y 581.199,Z 296.393,A -85,B 0,C 180,E1 -1912.39,E2 -1912.39} C_VEL
LIN {X 0,Y 581.423,Z 272.984,A -85,B 0,C 180,E1 -1915.219,E2 -1915.219} C_VEL
LIN {X 0,Y 580.876,Z 268.292,A -85,B 0,C 180,E1 -1915.821,E2 -1915.821} C_VEL
LIN {X 0,Y 580.282,Z 265.832,A -85,B 0,C 180,E1 -1916.172,E2 -1916.172} C_VEL
LIN {X 0,Y 580.295,Z 265.822,A -85,B 0,C 180,E1 -1919.308,E2 -1919.308} C_VEL
LIN {X 0,Y 580.294,Z 265.83,A -85,B 0,C 180,E1 -1922.2,E2 -1922.2} C_VEL
LIN {X 0,Y 580.273,Z 265.826,A -85,B 0,C 180,E1 -1924.697,E2 -1924.697} C_VEL
LIN {X 0,Y 580.271,Z 265.824,A -85,B 0,C 180,E1 -1927.27,E2 -1927.27} C_VEL
LIN {X 0,Y 580.282,Z 265.829,A -85,B 0,C 180,E1 -1930.269,E2 -1930.269} C_VEL
LIN {X 0,Y 580.249,Z 265.827,A -85,B 0,C 180,E1 -1932.708,E2 -1932.708} C_VEL
LIN {X 0,Y 580.248,Z 265.83,A -85,B 0,C 180,E1 -1935.61,E2 -1935.61} C_VEL
LIN {X 0,Y 580.248,Z 265.833,A -85,B 0,C 180,E1 -1938.228,E2 -1938.228} C_VEL
LIN {X 0,Y 580.259,Z 265.824,A -85,B 0,C 180,E1 -1940.963,E2 -1940.963} C_VEL
LIN {X 0,Y 580.235,Z 265.833,A -85,B 0,C 180,E1 -1943.593,E2 -1943.593} C_VEL
LIN {X 0,Y 580.273,Z 265.829,A -85,B 0,C 180,E1 -1946.142,E2 -1946.142} C_VEL
LIN {X 0,Y 580.261,Z 265.825,A -85,B 0,C 180,E1 -1948.613,E2 -1948.613} C_VEL
LIN {X 0,Y 580.279,Z 265.822,A -85,B 0,C 180,E1 -1951.022,E2 -1951.022} C_VEL
LIN {X 0,Y 580.238,Z 265.833,A -85,B 0,C 180,E1 -1954.148,E2 -1954.148} C_VEL
LIN {X 0,Y 580.256,Z 265.826,A -85,B 0,C 180,E1 -1956.44,E2 -1956.44} C_VEL
LIN {X 0,Y 580.26,Z 265.83,A -85,B 0,C 180,E1 -1959.436,E2 -1959.436} C_VEL
LIN {X 0,Y 580.236,Z 265.836,A -85,B 0,C 180,E1 -1961.643,E2 -1961.643} C_VEL
LIN {X 0,Y 580.269,Z 265.823,A -85,B 0,C 180,E1 -1964.546,E2 -1964.546} C_VEL
LIN {X 0,Y 580.239,Z 265.824,A -85,B 0,C 180,E1 -1966.694,E2 -1966.694} C_VEL
LIN {X 0,Y 580.26,Z 265.823,A -85,B 0,C 180,E1 -1968.825,E2 -1968.825} C_VEL
LIN {X 0,Y 580.281,Z 265.832,A -85,B 0,C 180,E1 -1971.642,E2 -1971.642} C_VEL
LIN {X 0,Y 580.252,Z 265.832,A -85,B 0,C 180,E1 -1973.741,E2 -1973.741} C_VEL
LIN {X 0,Y 580.233,Z 265.831,A -85,B 0,C 180,E1 -1975.831,E2 -1975.831} C_VEL
LIN {X 0,Y 580.305,Z 265.822,A -85,B 0,C 180,E1 -1977.917,E2 -1977.917} C_VEL
LIN {X 0,Y 580.316,Z 265.82,A -85,B 0,C 180,E1 -1979.999,E2 -1979.999} C_VEL
LIN {X 0,Y 580.296,Z 265.82,A -85,B 0,C 180,E1 -1982.776,E2 -1982.776} C_VEL
LIN {X 0,Y 580.292,Z 265.826,A -85,B 0,C 180,E1 -1985.559,E2 -1985.559} C_VEL
LIN {X 0,Y 580.265,Z 265.822,A -85,B 0,C 180,E1 -1988.356,E2 -1988.356} C_VEL
LIN {X 0,Y 580.29,Z 265.827,A -85,B 0,C 180,E1 -1991.19,E2 -1991.19} C_VEL
LIN {X 0,Y 580.254,Z 265.824,A -85,B 0,C 180,E1 -1994.318,E2 -1994.318} C_VEL
LIN {X 0,Y 580.254,Z 265.825,A -85,B 0,C 180,E1 -1996.898,E2 -1996.898} C_VEL
LIN {X 0,Y 580.258,Z 265.827,A -85,B 0,C 180,E1 -1999.822,E2 -1999.822} C_VEL
LIN {X 0,Y 580.272,Z 265.832,A -85,B 0,C 180,E1 -2001.276,E2 -2001.276} C_VEL
LIN {X 0,Y 579.555,Z 265.929,A -85,B 0,C 180,E1 -2001.855,E2 -2001.855} C_VEL
LIN {X 0,Y 576.667,Z 266.285,A -85,B 0,C 180,E1 -2002.795,E2 -2002.795} C_VEL
LIN {X 0,Y 574.266,Z 266.576,A -85,B 0,C 180,E1 -2003.551,E2 -2003.551} C_VEL
LIN {X 0,Y 573.254,Z 266.697,A -85,B 0,C 180,E1 -2004.135,E2 -2004.135} C_VEL
LIN {X 0,Y 573.18,Z 266.706,A -85,B 0,C 180,E1 -2004.332,E2 -2004.332} C_VEL
LIN {X 0,Y 573.182,Z 266.708,A -85,B 0,C 180,E1 -2006.978,E2 -2006.978} C_VEL
LIN {X 0,Y 573.198,Z 266.709,A -85,B 0,C 180,E1 -2009.481,E2 -2009.481} C_VEL
LIN {X 0,Y 573.231,Z 266.7,A -85,B 0,C 180,E1 -2012.226,E2 -2012.226} C_VEL
LIN {X 0,Y 573.207,Z 266.706,A -85,B 0,C 180,E1 -2014.768,E2 -2014.768} C_VEL
LIN {X 0,Y 573.21,Z 266.702,A -85,B 0,C 180,E1 -2017.807,E2 -2017.807} C_VEL
LIN {X 0,Y 573.228,Z 266.702,A -85,B 0,C 180,E1 -2020.524,E2 -2020.524} C_VEL
LIN {X 0,Y 573.218,Z 266.702,A -85,B 0,C 180,E1 -2023.667,E2 -2023.667} C_VEL
LIN {X 0,Y 573.191,Z 266.707,A -85,B 0,C 180,E1 -2026.637,E2 -2026.637} C_VEL
LIN {X 0,Y 573.226,Z 266.704,A -85,B 0,C 180,E1 -2029.474,E2 -2029.474} C_VEL
LIN {X 0,Y 573.213,Z 266.702,A -85,B 0,C 180,E1 -2032.191,E2 -2032.191} C_VEL
LIN {X 0,Y 573.223,Z 266.707,A -85,B 0,C 180,E1 -2035.227,E2 -2035.227} C_VEL
LIN {X 0,Y 573.225,Z 266.701,A -85,B 0,C 180,E1 -2038.184,E2 -2038.184} C_VEL
LIN {X 0,Y 573.237,Z 266.703,A -85,B 0,C 180,E1 -2040.633,E2 -2040.633} C_VEL
LIN {X 0,Y 573.231,Z 266.707,A -85,B 0,C 180,E1 -2043.023,E2 -2043.023} C_VEL
LIN {X 0,Y 573.253,Z 266.699,A -85,B 0,C 180,E1 -2045.365,E2 -2045.365} C_VEL
LIN {X 0,Y 573.207,Z 266.708,A -85,B 0,C 180,E1 -2048.419,E2 -2048.419} C_VEL
LIN {X 0,Y 573.259,Z 266.706,A -85,B 0,C 180,E1 -2050.728,E2 -2050.728} C_VEL
LIN {X 0,Y 573.227,Z 266.7,A -85,B 0,C 180,E1 -2053.621,E2 -2053.621} C_VEL
LIN {X 0,Y 573.246,Z 266.698,A -85,B 0,C 180,E1 -2055.806,E2 -2055.806} C_VEL
LIN {X 0,Y 573.271,Z 266.704,A -85,B 0,C 180,E1 -2058.73,E2 -2058.73} C_VEL
LIN {X 0,Y 573.236,Z 266.7,A -85,B 0,C 180,E1 -2061.54,E2 -2061.54} C_VEL
LIN {X 0,Y 573.275,Z 266.701,A -85,B 0,C 180,E1 -2064.372,E2 -2064.372} C_VEL
LIN {X 0,Y 573.288,Z 266.696,A -85,B 0,C 180,E1 -2067.189,E2 -2067.189} C_VEL
LIN {X 0,Y 573.293,Z 266.696,A -85,B 0,C 180,E1 -2070,E2 -2070} C_VEL
LIN {X 0,Y 573.3,Z 266.699,A -85,B 0,C 180,E1 -2072.81,E2 -2072.81} C_VEL
LIN {X 0,Y 573.269,Z 266.698,A -85,B 0,C 180,E1 -2075.628,E2 -2075.628} C_VEL
LIN {X 0,Y 573.307,Z 266.897,A -85,B 0,C 180,E1 -2076.783,E2 -2076.783} C_VEL
LIN {X 0,Y 574.066,Z 272.316,A -85,B 0,C 180,E1 -2077.58,E2 -2077.58} C_VEL
LIN {X 0,Y 573.872,Z 288.803,A -85,B 0,C 180,E1 -2079.872,E2 -2079.872} C_VEL
LIN {X 0,Y 573.819,Z 292.853,A -85,B 0,C 180,E1 -2080.43,E2 -2080.43} C_VEL
LIN {X 0,Y 575.175,Z 300.082,A -85,B 0,C 180,E1 -2080.583,E2 -2080.583} C_VEL
LIN {X 0,Y 574.723,Z 457.962,A -85,B 0,C 180,E1 -2082.625,E2 -2082.625} C_VEL
LIN {X 0,Y 574.615,Z 473.244,A -85,B 0,C 180,E1 -2082.965,E2 -2082.965} C_VEL
LIN {X 0,Y 574.426,Z 488.155,A -85,B 0,C 180,E1 -2083.441,E2 -2083.441} C_VEL
LIN {X 0,Y 574.229,Z 503.087,A -85,B 0,C 180,E1 -2084.078,E2 -2084.078} C_VEL
LIN {X 0,Y 574.024,Z 516.704,A -85,B 0,C 180,E1 -2084.811,E2 -2084.811} C_VEL
LIN {X 0,Y 573.853,Z 529.165,A -85,B 0,C 180,E1 -2085.63,E2 -2085.63} C_VEL
LIN {X 0,Y 573.646,Z 541.943,A -85,B 0,C 180,E1 -2086.641,E2 -2086.641} C_VEL
LIN {X 0,Y 573.459,Z 552.715,A -85,B 0,C 180,E1 -2087.656,E2 -2087.656} C_VEL
LIN {X 0,Y 573.345,Z 562.68,A -85,B 0,C 180,E1 -2088.767,E2 -2088.767} C_VEL
LIN {X 0,Y 573.226,Z 572.514,A -85,B 0,C 180,E1 -2090.077,E2 -2090.077} C_VEL
LIN {X 0,Y 573.118,Z 579.939,A -85,B 0,C 180,E1 -2091.262,E2 -2091.262} C_VEL
LIN {X 0,Y 573.062,Z 587.455,A -85,B 0,C 180,E1 -2092.725,E2 -2092.725} C_VEL
LIN {X 0,Y 573.023,Z 593.624,A -85,B 0,C 180,E1 -2094.259,E2 -2094.259} C_VEL
LIN {X 0,Y 572.995,Z 597.273,A -85,B 0,C 180,E1 -2095.421,E2 -2095.421} C_VEL
LIN {X 0,Y 572.934,Z 600.804,A -85,B 0,C 180,E1 -2096.991,E2 -2096.991} C_VEL
LIN {X 0,Y 572.92,Z 602.872,A -85,B 0,C 180,E1 -2098.581,E2 -2098.581} C_VEL
LIN {X 0,Y 572.956,Z 603.372,A -85,B 0,C 180,E1 -2099.441,E2 -2099.441} C_VEL
LIN {X 0,Y 572.946,Z 603.207,A -85,B 0,C 180,E1 -2101.009,E2 -2101.009} C_VEL
LIN {X 0,Y 572.937,Z 602.161,A -85,B 0,C 180,E1 -2102.182,E2 -2102.182} C_VEL
LIN {X 0,Y 572.966,Z 600.01,A -85,B 0,C 180,E1 -2103.501,E2 -2103.501} C_VEL
LIN {X 0,Y 572.987,Z 597.073,A -85,B 0,C 180,E1 -2104.739,E2 -2104.739} C_VEL
LIN {X 0,Y 573.029,Z 592.808,A -85,B 0,C 180,E1 -2106.064,E2 -2106.064} C_VEL
LIN {X 0,Y 573.035,Z 587.052,A -85,B 0,C 180,E1 -2107.454,E2 -2107.454} C_VEL
LIN {X 0,Y 573.112,Z 579.588,A -85,B 0,C 180,E1 -2108.89,E2 -2108.89} C_VEL
LIN {X 0,Y 573.194,Z 572.149,A -85,B 0,C 180,E1 -2110.067,E2 -2110.067} C_VEL
LIN {X 0,Y 573.338,Z 563.583,A -85,B 0,C 180,E1 -2111.212,E2 -2111.212} C_VEL
LIN {X 0,Y 573.452,Z 553.24,A -85,B 0,C 180,E1 -2112.38,E2 -2112.38} C_VEL
LIN {X 0,Y 573.621,Z 541.077,A -85,B 0,C 180,E1 -2113.525,E2 -2113.525} C_VEL
LIN {X 0,Y 573.855,Z 528.434,A -85,B 0,C 180,E1 -2114.513,E2 -2114.513} C_VEL
LIN {X 0,Y 574.051,Z 515.609,A -85,B 0,C 180,E1 -2115.343,E2 -2115.343} C_VEL
LIN {X 0,Y 574.265,Z 501.604,A -85,B 0,C 180,E1 -2116.083,E2 -2116.083} C_VEL
LIN {X 0,Y 574.462,Z 487.501,A -85,B 0,C 180,E1 -2116.672,E2 -2116.672} C_VEL
LIN {X 0,Y 574.628,Z 472.533,A -85,B 0,C 180,E1 -2117.144,E2 -2117.144} C_VEL
LIN {X 0,Y 574.743,Z 456.669,A -85,B 0,C 180,E1 -2117.487,E2 -2117.487} C_VEL
LIN {X 0,Y 575.161,Z 299.434,A -85,B 0,C 180,E1 -2119.516,E2 -2119.516} C_VEL
LIN {X 0,Y 573.828,Z 292.774,A -85,B 0,C 180,E1 -2119.671,E2 -2119.671} C_VEL
LIN {X 0,Y 574.078,Z 273.01,A -85,B 0,C 180,E1 -2122.412,E2 -2122.412} C_VEL
LIN {X 0,Y 573.569,Z 268.256,A -85,B 0,C 180,E1 -2123.104,E2 -2123.104} C_VEL
LIN {X 0,Y 573.271,Z 266.705,A -85,B 0,C 180,E1 -2123.355,E2 -2123.355} C_VEL
LIN {X 0,Y 573.269,Z 266.698,A -85,B 0,C 180,E1 -2126.473,E2 -2126.473} C_VEL
LIN {X 0,Y 573.228,Z 266.706,A -85,B 0,C 180,E1 -2129.115,E2 -2129.115} C_VEL
LIN {X 0,Y 573.248,Z 266.701,A -85,B 0,C 180,E1 -2131.969,E2 -2131.969} C_VEL
LIN {X 0,Y 573.24,Z 266.7,A -85,B 0,C 180,E1 -2134.591,E2 -2134.591} C_VEL
LIN {X 0,Y 573.224,Z 266.706,A -85,B 0,C 180,E1 -2137.663,E2 -2137.663} C_VEL
LIN {X 0,Y 573.242,Z 266.701,A -85,B 0,C 180,E1 -2139.925,E2 -2139.925} C_VEL
LIN {X 0,Y 573.246,Z 266.705,A -85,B 0,C 180,E1 -2142.99,E2 -2142.99} C_VEL
LIN {X 0,Y 573.258,Z 266.699,A -85,B 0,C 180,E1 -2145.808,E2 -2145.808} C_VEL
LIN {X 0,Y 573.247,Z 266.703,A -85,B 0,C 180,E1 -2148.746,E2 -2148.746} C_VEL
LIN {X 0,Y 573.24,Z 266.702,A -85,B 0,C 180,E1 -2151.541,E2 -2151.541} C_VEL
LIN {X 0,Y 573.221,Z 266.703,A -85,B 0,C 180,E1 -2153.666,E2 -2153.666} C_VEL
LIN {X 0,Y 573.201,Z 266.704,A -85,B 0,C 180,E1 -2155.782,E2 -2155.782} C_VEL
LIN {X 0,Y 573.284,Z 266.694,A -85,B 0,C 180,E1 -2157.894,E2 -2157.894} C_VEL
LIN {X 0,Y 573.329,Z 266.695,A -85,B 0,C 180,E1 -2160.704,E2 -2160.704} C_VEL
LIN {X 0,Y 573.206,Z 266.705,A -85,B 0,C 180,E1 -2163.516,E2 -2163.516} C_VEL
LIN {X 0,Y 573.262,Z 266.697,A -85,B 0,C 180,E1 -2165.63,E2 -2165.63} C_VEL
LIN {X 0,Y 573.227,Z 266.7,A -85,B 0,C 180,E1 -2167.752,E2 -2167.752} C_VEL
LIN {X 0,Y 573.254,Z 266.705,A -85,B 0,C 180,E1 -2170.598,E2 -2170.598} C_VEL
LIN {X 0,Y 573.208,Z 266.703,A -85,B 0,C 180,E1 -2173.472,E2 -2173.472} C_VEL
LIN {X 0,Y 573.216,Z 266.702,A -85,B 0,C 180,E1 -2175.649,E2 -2175.649} C_VEL
LIN {X 0,Y 573.226,Z 266.701,A -85,B 0,C 180,E1 -2177.85,E2 -2177.85} C_VEL
LIN {X 0,Y 573.227,Z 266.703,A -85,B 0,C 180,E1 -2180.078,E2 -2180.078} C_VEL
LIN {X 0,Y 573.216,Z 266.709,A -85,B 0,C 180,E1 -2182.339,E2 -2182.339} C_VEL
LIN {X 0,Y 573.198,Z 266.708,A -85,B 0,C 180,E1 -2184.866,E2 -2184.866} C_VEL
LIN {X 0,Y 573.222,Z 266.703,A -85,B 0,C 180,E1 -2187.769,E2 -2187.769} C_VEL
LIN {X 0,Y 573.213,Z 266.709,A -85,B 0,C 180,E1 -2190.179,E2 -2190.179} C_VEL
LIN {X 0,Y 573.235,Z 266.705,A -85,B 0,C 180,E1 -2192.647,E2 -2192.647} C_VEL
LIN {X 0,Y 573.172,Z 266.708,A -85,B 0,C 180,E1 -2195.191,E2 -2195.191} C_VEL
LIN {X 0,Y 573.207,Z 266.706,A -85,B 0,C 180,E1 -2197.81,E2 -2197.81} C_VEL
LIN {X 0,Y 573.195,Z 266.709,A -85,B 0,C 180,E1 -2200.53,E2 -2200.53} C_VEL
LIN {X 0,Y 573.192,Z 266.706,A -85,B 0,C 180,E1 -2203.364,E2 -2203.364} C_VEL
LIN {X 0,Y 573.196,Z 266.711,A -85,B 0,C 180,E1 -2206.337,E2 -2206.337} C_VEL
LIN {X 0,Y 573.24,Z 266.702,A -85,B 0,C 180,E1 -2209.476,E2 -2209.476} C_VEL
LIN {X 0,Y 573.215,Z 266.708,A -85,B 0,C 180,E1 -2212.192,E2 -2212.192} C_VEL
LIN {X 0,Y 573.217,Z 266.704,A -85,B 0,C 180,E1 -2215.232,E2 -2215.232} C_VEL
LIN {X 0,Y 573.243,Z 266.708,A -85,B 0,C 180,E1 -2217.774,E2 -2217.774} C_VEL
LIN {X 0,Y 573.256,Z 266.7,A -85,B 0,C 180,E1 -2220.635,E2 -2220.635} C_VEL
LIN {X 0,Y 573.258,Z 266.899,A -85,B 0,C 180,E1 -2223.664,E2 -2223.664} C_VEL
LIN {X 0,Y 574.574,Z 272.866,A -85,B 0,C 180,E1 -2224.459,E2 -2224.459} C_VEL
LIN {X 0,Y 574.388,Z 291.328,A -85,B 0,C 180,E1 -2226.712,E2 -2226.712} C_VEL
LIN {X 0,Y 574.085,Z 313.565,A -85,B 0,C 180,E1 -2229.394,E2 -2229.394} C_VEL
LIN {X 0,Y 574.014,Z 321.877,A -85,B 0,C 180,E1 -2230.386,E2 -2230.386} C_VEL
LIN {X 0,Y 575.177,Z 328.502,A -85,B 0,C 180,E1 -2230.517,E2 -2230.517} C_VEL
LIN {X 0,Y 574.766,Z 487.977,A -85,B 0,C 180,E1 -2232.579,E2 -2232.579} C_VEL
LIN {X 0,Y 574.633,Z 503.729,A -85,B 0,C 180,E1 -2232.931,E2 -2232.931} C_VEL
LIN {X 0,Y 574.411,Z 519.057,A -85,B 0,C 180,E1 -2233.428,E2 -2233.428} C_VEL
LIN {X 0,Y 574.292,Z 532.785,A -85,B 0,C 180,E1 -2234.018,E2 -2234.018} C_VEL
LIN {X 0,Y 574.048,Z 546.255,A -85,B 0,C 180,E1 -2234.739,E2 -2234.739} C_VEL
LIN {X 0,Y 573.86,Z 559.828,A -85,B 0,C 180,E1 -2235.632,E2 -2235.632} C_VEL
LIN {X 0,Y 573.635,Z 572.357,A -85,B 0,C 180,E1 -2236.63,E2 -2236.63} C_VEL
LIN {X 0,Y 573.477,Z 582.755,A -85,B 0,C 180,E1 -2237.617,E2 -2237.617} C_VEL
LIN {X 0,Y 573.286,Z 592.774,A -85,B 0,C 180,E1 -2238.735,E2 -2238.735} C_VEL
LIN {X 0,Y 573.243,Z 601.861,A -85,B 0,C 180,E1 -2239.939,E2 -2239.939} C_VEL
LIN {X 0,Y 573.133,Z 609.736,A -85,B 0,C 180,E1 -2241.183,E2 -2241.183} C_VEL
LIN {X 0,Y 573.075,Z 617.091,A -85,B 0,C 180,E1 -2242.602,E2 -2242.602} C_VEL
LIN {X 0,Y 573.04,Z 622.924,A -85,B 0,C 180,E1 -2244.017,E2 -2244.017} C_VEL
LIN {X 0,Y 572.951,Z 626.386,A -85,B 0,C 180,E1 -2245.075,E2 -2245.075} C_VEL
